gfCNCPoint2[15649] = {X 94.9398, Y 8.2871, Z -3.0000, A 0.000, B 0.000, C 0.000 }
gfCNCPoint2[15650] = {X 95.7852, Y 8.5829, Z -3.0000, A 0.000, B 0.000, C 0.000 }
gfCNCPoint2[15651] = {X 96.5436, Y 9.0595, Z -3.0000, A 0.000, B 0.000, C 0.000 }
gfCNCPoint2[15652] = {X 97.1770, Y 9.6929, Z -3.0000, A 0.000, B 0.000, C 0.000 }
gfCNCPoint2[15653] = {X 97.6535, Y 10.4513, Z -3.0000, A 0.000, B 0.000, C 0.000 }
gfCNCPoint2[15654] = {X 97.9494, Y 11.2967, Z -3.0000, A 0.000, B 0.000, C 0.000 }
gfCNCPoint2[15655] = {X 98.0497, Y 12.1868, Z -3.0000, A 0.000, B 0.000, C 0.000 }
gfCNCPoint2[15656] = {X 98.0495, Y 13.0192, Z -3.0000, A 0.000, B 0.000, C 0.000 }
gfCNCPoint2[15657] = {X 97.9794, Y 13.7247, Z -3.0000, A 0.000, B 0.000, C 0.000 }
gfCNCPoint2[15658] = {X 97.7858, Y 14.4068, Z -3.0000, A 0.000, B 0.000, C 0.000 }
gfCNCPoint2[15659] = {X 97.4749, Y 15.0440, Z -3.0000, A 0.000, B 0.000, C 0.000 }
gfCNCPoint2[15660] = {X 97.4127, Y 15.1437, Z -3.0000, A 0.000, B 0.000, C 0.000 }
gfCNCPoint2[15661] = {X 97.3476, Y 15.2415, Z -3.0000, A 0.000, B 0.000, C 0.000 }
gfCNCPoint2[15662] = {X 97.4105, Y 15.3108, Z -3.0000, A 0.000, B 0.000, C 0.000 }
gfCNCPoint2[15663] = {X 97.9961, Y 16.7687, Z -3.0000, A 0.000, B 0.000, C 0.000 }
gfCNCPoint2[15664] = {X 101.6269, Y 25.7689, Z -3.0000, A 0.000, B 0.000, C 0.000 }
gfCNCPoint2[15665] = {X 101.8768, Y 26.3801, Z -3.0000, A 0.000, B 0.000, C 0.000 }
gfCNCPoint2[15666] = {X 102.1268, Y 25.7689, Z -3.0000, A 0.000, B 0.000, C 0.000 }
gfCNCPoint2[15667] = {X 106.3426, Y 15.2553, Z -3.0000, A 0.000, B 0.000, C 0.000 }
gfCNCPoint2[15668] = {X 106.3813, Y 15.1986, Z -3.0000, A 0.000, B 0.000, C 0.000 }
gfCNCPoint2[15669] = {X 106.3236, Y 15.1097, Z -3.0000, A 0.000, B 0.000, C 0.000 }
gfCNCPoint2[15670] = {X 106.2684, Y 15.0194, Z -3.0000, A 0.000, B 0.000, C 0.000 }
gfCNCPoint2[15671] = {X 105.9605, Y 14.3760, Z -3.0000, A 0.000, B 0.000, C 0.000 }
gfCNCPoint2[15672] = {X 105.7718, Y 13.6883, Z -3.0000, A 0.000, B 0.000, C 0.000 }
gfCNCPoint2[15673] = {X 105.7083, Y 12.9779, Z -3.0000, A 0.000, B 0.000, C 0.000 }
gfCNCPoint2[15674] = {X 105.7083, Y 12.1868, Z -3.0000, A 0.000, B 0.000, C 0.000 }
gfCNCPoint2[15675] = {X 105.8086, Y 11.2967, Z -3.0000, A 0.000, B 0.000, C 0.000 }
gfCNCPoint2[15676] = {X 106.1044, Y 10.4513, Z -3.0000, A 0.000, B 0.000, C 0.000 }
gfCNCPoint2[15677] = {X 106.5810, Y 9.6929, Z -3.0000, A 0.000, B 0.000, C 0.000 }
gfCNCPoint2[15678] = {X 107.2143, Y 9.0595, Z -3.0000, A 0.000, B 0.000, C 0.000 }
gfCNCPoint2[15679] = {X 107.9727, Y 8.5829, Z -3.0000, A 0.000, B 0.000, C 0.000 }
gfCNCPoint2[15680] = {X 108.8182, Y 8.2871, Z -3.0000, A 0.000, B 0.000, C 0.000 }
gfCNCPoint2[15681] = {X 109.7083, Y 8.1868, Z -3.0000, A 0.000, B 0.000, C 0.000 }
gfCNCPoint2[15682] = {X 117.7916, Y 8.1868, Z -3.0000, A 0.000, B 0.000, C 0.000 }
gfCNCPoint2[15683] = {X 118.6817, Y 8.2871, Z -3.0000, A 0.000, B 0.000, C 0.000 }
gfCNCPoint2[15684] = {X 119.5271, Y 8.5829, Z -3.0000, A 0.000, B 0.000, C 0.000 }
gfCNCPoint2[15685] = {X 120.2855, Y 9.0595, Z -3.0000, A 0.000, B 0.000, C 0.000 }
gfCNCPoint2[15686] = {X 120.9189, Y 9.6929, Z -3.0000, A 0.000, B 0.000, C 0.000 }
gfCNCPoint2[15687] = {X 121.3955, Y 10.4513, Z -3.0000, A 0.000, B 0.000, C 0.000 }
gfCNCPoint2[15688] = {X 121.6913, Y 11.2967, Z -3.0000, A 0.000, B 0.000, C 0.000 }
gfCNCPoint2[15689] = {X 121.7916, Y 12.1868, Z -3.0000, A 0.000, B 0.000, C 0.000 }
gfCNCPoint2[15690] = {X 121.7914, Y 13.0192, Z -3.0000, A 0.000, B 0.000, C 0.000 }
gfCNCPoint2[15691] = {X 121.6828, Y 13.9047, Z -3.0000, A 0.000, B 0.000, C 0.000 }
gfCNCPoint2[15692] = {X 121.3806, Y 14.7440, Z -3.0000, A 0.000, B 0.000, C 0.000 }
gfCNCPoint2[15693] = {X 120.9000, Y 15.4955, Z -3.0000, A 0.000, B 0.000, C 0.000 }
gfCNCPoint2[15694] = {X 120.2647, Y 16.1219, Z -3.0000, A 0.000, B 0.000, C 0.000 }
gfCNCPoint2[15695] = {X 120.2634, Y 41.0662, Z -3.0000, A 0.000, B 0.000, C 0.000 }
gfCNCPoint2[15696] = {X 120.4160, Y 41.1901, Z -3.0000, A 0.000, B 0.000, C 0.000 }
gfCNCPoint2[15697] = {X 120.9967, Y 41.8157, Z -3.0000, A 0.000, B 0.000, C 0.000 }
gfCNCPoint2[15698] = {X 121.4315, Y 42.5502, Z -3.0000, A 0.000, B 0.000, C 0.000 }
gfCNCPoint2[15699] = {X 121.7005, Y 43.3602, Z -3.0000, A 0.000, B 0.000, C 0.000 }
gfCNCPoint2[15700] = {X 121.7916, Y 44.2089, Z -3.0000, A 0.000, B 0.000, C 0.000 }
gfCNCPoint2[15701] = {X 121.7916, Y 45.0000, Z -3.0000, A 0.000, B 0.000, C 0.000 }
gfCNCPoint2[15702] = {X 121.6913, Y 45.8901, Z -3.0000, A 0.000, B 0.000, C 0.000 }
gfCNCPoint2[15703] = {X 121.3955, Y 46.7355, Z -3.0000, A 0.000, B 0.000, C 0.000 }
gfCNCPoint2[15704] = {X 120.9189, Y 47.4940, Z -3.0000, A 0.000, B 0.000, C 0.000 }
gfCNCPoint2[15705] = {X 120.2855, Y 48.1273, Z -3.0000, A 0.000, B 0.000, C 0.000 }
gfCNCPoint2[15706] = {X 119.5271, Y 48.6039, Z -3.0000, A 0.000, B 0.000, C 0.000 }
gfCNCPoint2[15707] = {X 118.6817, Y 48.8997, Z -3.0000, A 0.000, B 0.000, C 0.000 }
gfCNCPoint2[15708] = {X 117.7916, Y 49.0000, Z -3.0000, A 0.000, B 0.000, C 0.000 }
gfCNCPoint2[15709] = {X 111.9185, Y 49.0000, Z -3.0000, A 0.000, B 0.000, C 0.000 }
gfCNCPoint2[15710] = {X 111.0284, Y 48.8997, Z -3.0000, A 0.000, B 0.000, C 0.000 }
gfCNCPoint2[15711] = {X 110.1829, Y 48.6039, Z -3.0000, A 0.000, B 0.000, C 0.000 }
gfCNCPoint2[15712] = {X 109.4245, Y 48.1273, Z -3.0000, A 0.000, B 0.000, C 0.000 }
gfCNCPoint2[15713] = {X 108.7911, Y 47.4939, Z -3.0000, A 0.000, B 0.000, C 0.000 }
gfCNCPoint2[15714] = {X 108.3146, Y 46.7355, Z -3.0000, A 0.000, B 0.000, C 0.000 }
gfCNCPoint2[15715] = {X 108.0188, Y 45.8900, Z -3.0000, A 0.000, B 0.000, C 0.000 }
gfCNCPoint2[15716] = {X 107.9185, Y 45.0000, Z -3.0000, A 0.000, B 0.000, C 0.000 }
gfCNCPoint2[15717] = {X 107.9185, Y 44.1811, Z -3.0000, A 0.000, B 0.000, C 0.000 }
gfCNCPoint2[15718] = {X 107.9517, Y 43.6776, Z -3.0000, A 0.000, B 0.000, C 0.000 }
gfCNCPoint2[15719] = {X 108.0507, Y 43.1827, Z -3.0000, A 0.000, B 0.000, C 0.000 }
gfCNCPoint2[15720] = {X 108.2043, Y 42.7280, Z -3.0000, A 0.000, B 0.000, C 0.000 }
gfCNCPoint2[15721] = {X 108.4135, Y 42.2960, Z -3.0000, A 0.000, B 0.000, C 0.000 }
gfCNCPoint2[15722] = {X 108.4390, Y 42.2514, Z -3.0000, A 0.000, B 0.000, C 0.000 }
gfCNCPoint2[15723] = {X 108.4651, Y 42.2073, Z -3.0000, A 0.000, B 0.000, C 0.000 }
gfCNCPoint2[15724] = {X 108.9129, Y 41.5686, Z -3.0000, A 0.000, B 0.000, C 0.000 }
gfCNCPoint2[15725] = {X 109.4466, Y 40.9999, Z -3.0000, A 0.000, B 0.000, C 0.000 }
gfCNCPoint2[15726] = {X 109.4465, Y 38.9229, Z -3.0000, A 0.000, B 0.000, C 0.000 }
gfCNCPoint2[15727] = {X 108.9328, Y 38.9229, Z -3.0000, A 0.000, B 0.000, C 0.000 }
gfCNCPoint2[15728] = {X 105.8164, Y 46.5384, Z -3.0000, A 0.000, B 0.000, C 0.000 }
gfCNCPoint2[15729] = {X 105.3339, Y 47.3869, Z -3.0000, A 0.000, B 0.000, C 0.000 }
gfCNCPoint2[15730] = {X 104.6602, Y 48.0932, Z -3.0000, A 0.000, B 0.000, C 0.000 }
gfCNCPoint2[15731] = {X 103.8355, Y 48.6154, Z -3.0000, A 0.000, B 0.000, C 0.000 }
gfCNCPoint2[15732] = {X 102.9580, Y 48.9121, Z -3.0000, A 0.000, B 0.000, C 0.000 }
gfCNCPoint2[15733] = {X 102.0357, Y 48.9990, Z -3.0000, A 0.000, B 0.000, C 0.000 }
gfCNCPoint2[15734] = {X 101.1182, Y 48.8715, Z -3.0000, A 0.000, B 0.000, C 0.000 }
gfCNCPoint2[15735] = {X 100.2546, Y 48.5362, Z -3.0000, A 0.000, B 0.000, C 0.000 }
gfCNCPoint2[15736] = {X 99.4912, Y 48.0114, Z -3.0000, A 0.000, B 0.000, C 0.000 }
gfCNCPoint2[15737] = {X 98.8691, Y 47.3250, Z -3.0000, A 0.000, B 0.000, C 0.000 }
gfCNCPoint2[15738] = {X 98.4216, Y 46.5139, Z -3.0000, A 0.000, B 0.000, C 0.000 }
gfCNCPoint2[15739] = {X 94.8150, Y 37.6933, Z -3.0000, A 0.000, B 0.000, C 0.000 }
gfCNCPoint2[15740] = {X 94.8103, Y 38.2306, Z -3.0000, A 0.000, B 0.000, C 0.000 }
gfCNCPoint2[15741] = {X 94.8105, Y 41.0553, Z -3.0000, A 0.000, B 0.000, C 0.000 }
gfCNCPoint2[15742] = {X 95.3658, Y 41.5952, Z -3.0000, A 0.000, B 0.000, C 0.000 }
gfCNCPoint2[15743] = {X 95.8092, Y 42.2301, Z -3.0000, A 0.000, B 0.000, C 0.000 }
gfCNCPoint2[15744] = {X 96.0347, Y 42.6952, Z -3.0000, A 0.000, B 0.000, C 0.000 }
gfCNCPoint2[15745] = {X 96.1997, Y 43.1852, Z -3.0000, A 0.000, B 0.000, C 0.000 }
gfCNCPoint2[15746] = {X 96.3016, Y 43.6926, Z -3.0000, A 0.000, B 0.000, C 0.000 }
gfCNCPoint2[15747] = {X 96.3385, Y 44.2089, Z -3.0000, A 0.000, B 0.000, C 0.000 }
gfCNCPoint2[15748] = {X 96.3384, Y 45.0384, Z -3.0000, A 0.000, B 0.000, C 0.000 }
gfCNCPoint2[15749] = {X 96.2308, Y 45.9222, Z -3.0000, A 0.000, B 0.000, C 0.000 }
gfCNCPoint2[15750] = {X 95.9304, Y 46.7602, Z -3.0000, A 0.000, B 0.000, C 0.000 }
gfCNCPoint2[15751] = {X 95.4521, Y 47.5111, Z -3.0000, A 0.000, B 0.000, C 0.000 }
gfCNCPoint2[15752] = {X 94.8196, Y 48.1376, Z -3.0000, A 0.000, B 0.000, C 0.000 }
gfCNCPoint2[15753] = {X 94.0642, Y 48.6086, Z -3.0000, A 0.000, B 0.000, C 0.000 }
gfCNCPoint2[15754] = {X 93.2233, Y 48.9009, Z -3.0000, A 0.000, B 0.000, C 0.000 }
gfCNCPoint2[15755] = {X 92.3385, Y 49.0000, Z -3.0000, A 0.000, B 0.000, C 0.000 }
gfCNCPoint2[15756] = {X 85.8951, Y 49.0000, Z -3.0000, A 0.000, B 0.000, C 0.000 }
gfCNCPoint2[15757] = {X 85.0050, Y 48.8997, Z -3.0000, A 0.000, B 0.000, C 0.000 }
gfCNCPoint2[15758] = {X 84.1595, Y 48.6039, Z -3.0000, A 0.000, B 0.000, C 0.000 }
gfCNCPoint2[15759] = {X 83.4011, Y 48.1273, Z -3.0000, A 0.000, B 0.000, C 0.000 }
gfCNCPoint2[15760] = {X 82.7677, Y 47.4939, Z -3.0000, A 0.000, B 0.000, C 0.000 }
gfCNCPoint2[15761] = {X 82.2912, Y 46.7355, Z -3.0000, A 0.000, B 0.000, C 0.000 }
gfCNCPoint2[15762] = {X 81.9954, Y 45.8900, Z -3.0000, A 0.000, B 0.000, C 0.000 }
gfCNCPoint2[15763] = {X 81.8951, Y 45.0000, Z -3.0000, A 0.000, B 0.000, C 0.000 }
gfCNCPoint2[15764] = {X 81.8951, Y 44.2089, Z -3.0000, A 0.000, B 0.000, C 0.000 }
gfCNCPoint2[15765] = {X 82.0011, Y 43.3123, Z -3.0000, A 0.000, B 0.000, C 0.000 }
gfCNCPoint2[15766] = {X 82.3025, Y 42.4613, Z -3.0000, A 0.000, B 0.000, C 0.000 }
gfCNCPoint2[15767] = {X 82.7846, Y 41.6979, Z -3.0000, A 0.000, B 0.000, C 0.000 }
gfCNCPoint2[15768] = {X 83.4234, Y 41.0598, Z -3.0000, A 0.000, B 0.000, C 0.000 }
gfCNCPoint2[15769] = {X 83.4233, Y 28.5920, Z -3.0000, A 0.000, B 0.000, C 0.000 }
gfCNCPoint2[15770] = {X 79.3433, Y 28.5920, Z -3.0000, A 0.000, B 0.000, C 0.000 }
gfCNCPoint2[15771] = {X 79.3433, Y 28.5920, Z 0.0000, A 0.000, B 0.000, C 0.000 }
gfCNCPoint2[15772] = {X 79.3433, Y 28.5920, Z 11.0000, A 0.000, B 0.000, C 0.000 }
gfCNCPoint2[15773] = {X 136.1636, Y 30.3963, Z 11.0000, A 0.000, B 0.000, C 0.000 }
gfCNCPoint2[15774] = {X 136.1636, Y 30.3963, Z 0.0000, A 0.000, B 0.000, C 0.000 }
gfCNCPoint2[15775] = {X 136.1636, Y 30.3963, Z -3.0000, A 0.000, B 0.000, C 0.000 }
gfCNCPoint2[15776] = {X 140.2436, Y 30.3963, Z -3.0000, A 0.000, B 0.000, C 0.000 }
gfCNCPoint2[15777] = {X 140.2436, Y 19.8770, Z -3.0000, A 0.000, B 0.000, C 0.000 }
gfCNCPoint2[15778] = {X 137.4242, Y 19.8766, Z -3.0000, A 0.000, B 0.000, C 0.000 }
gfCNCPoint2[15779] = {X 136.8918, Y 20.5215, Z -3.0000, A 0.000, B 0.000, C 0.000 }
gfCNCPoint2[15780] = {X 136.2452, Y 21.0516, Z -3.0000, A 0.000, B 0.000, C 0.000 }
gfCNCPoint2[15781] = {X 135.5085, Y 21.4473, Z -3.0000, A 0.000, B 0.000, C 0.000 }
gfCNCPoint2[15782] = {X 134.7094, Y 21.6936, Z -3.0000, A 0.000, B 0.000, C 0.000 }
gfCNCPoint2[15783] = {X 133.8778, Y 21.7814, Z -3.0000, A 0.000, B 0.000, C 0.000 }
gfCNCPoint2[15784] = {X 133.2006, Y 21.7815, Z -3.0000, A 0.000, B 0.000, C 0.000 }
gfCNCPoint2[15785] = {X 132.2394, Y 21.6732, Z -3.0000, A 0.000, B 0.000, C 0.000 }
gfCNCPoint2[15786] = {X 131.3263, Y 21.3537, Z -3.0000, A 0.000, B 0.000, C 0.000 }
gfCNCPoint2[15787] = {X 130.5072, Y 20.8390, Z -3.0000, A 0.000, B 0.000, C 0.000 }
gfCNCPoint2[15788] = {X 129.8231, Y 20.1550, Z -3.0000, A 0.000, B 0.000, C 0.000 }
gfCNCPoint2[15789] = {X 129.3085, Y 19.3359, Z -3.0000, A 0.000, B 0.000, C 0.000 }
gfCNCPoint2[15790] = {X 128.9890, Y 18.4228, Z -3.0000, A 0.000, B 0.000, C 0.000 }
gfCNCPoint2[15791] = {X 128.8806, Y 17.4615, Z -3.0000, A 0.000, B 0.000, C 0.000 }
gfCNCPoint2[15792] = {X 128.8806, Y 10.4835, Z -3.0000, A 0.000, B 0.000, C 0.000 }
gfCNCPoint2[15793] = {X 128.9874, Y 9.5289, Z -3.0000, A 0.000, B 0.000, C 0.000 }
gfCNCPoint2[15794] = {X 129.3026, Y 8.6214, Z -3.0000, A 0.000, B 0.000, C 0.000 }
gfCNCPoint2[15795] = {X 129.8104, Y 7.8061, Z -3.0000, A 0.000, B 0.000, C 0.000 }
gfCNCPoint2[15796] = {X 130.4859, Y 7.1231, Z -3.0000, A 0.000, B 0.000, C 0.000 }
gfCNCPoint2[15797] = {X 131.2956, Y 6.6063, Z -3.0000, A 0.000, B 0.000, C 0.000 }
gfCNCPoint2[15798] = {X 132.1995, Y 6.2811, Z -3.0000, A 0.000, B 0.000, C 0.000 }
gfCNCPoint2[15799] = {X 133.1529, Y 6.1638, Z -3.0000, A 0.000, B 0.000, C 0.000 }
gfCNCPoint2[15800] = {X 133.8866, Y 6.1637, Z -3.0000, A 0.000, B 0.000, C 0.000 }
gfCNCPoint2[15801] = {X 134.7112, Y 6.2518, Z -3.0000, A 0.000, B 0.000, C 0.000 }
gfCNCPoint2[15802] = {X 135.5038, Y 6.4958, Z -3.0000, A 0.000, B 0.000, C 0.000 }
gfCNCPoint2[15803] = {X 136.2352, Y 6.8868, Z -3.0000, A 0.000, B 0.000, C 0.000 }
gfCNCPoint2[15804] = {X 136.8784, Y 7.4103, Z -3.0000, A 0.000, B 0.000, C 0.000 }
gfCNCPoint2[15805] = {X 137.4097, Y 8.0470, Z -3.0000, A 0.000, B 0.000, C 0.000 }
gfCNCPoint2[15806] = {X 155.1123, Y 8.0482, Z -3.0000, A 0.000, B 0.000, C 0.000 }
gfCNCPoint2[15807] = {X 155.6443, Y 7.4103, Z -3.0000, A 0.000, B 0.000, C 0.000 }
gfCNCPoint2[15808] = {X 156.2886, Y 6.8861, Z -3.0000, A 0.000, B 0.000, C 0.000 }
gfCNCPoint2[15809] = {X 157.0212, Y 6.4948, Z -3.0000, A 0.000, B 0.000, C 0.000 }
gfCNCPoint2[15810] = {X 157.8152, Y 6.2510, Z -3.0000, A 0.000, B 0.000, C 0.000 }
gfCNCPoint2[15811] = {X 158.6412, Y 6.1637, Z -3.0000, A 0.000, B 0.000, C 0.000 }
gfCNCPoint2[15812] = {X 159.3781, Y 6.1639, Z -3.0000, A 0.000, B 0.000, C 0.000 }
gfCNCPoint2[15813] = {X 160.3301, Y 6.2828, Z -3.0000, A 0.000, B 0.000, C 0.000 }
gfCNCPoint2[15814] = {X 161.2324, Y 6.6088, Z -3.0000, A 0.000, B 0.000, C 0.000 }
gfCNCPoint2[15815] = {X 162.0405, Y 7.1260, Z -3.0000, A 0.000, B 0.000, C 0.000 }
gfCNCPoint2[15816] = {X 162.7145, Y 7.8088, Z -3.0000, A 0.000, B 0.000, C 0.000 }
gfCNCPoint2[15817] = {X 163.2212, Y 8.6236, Z -3.0000, A 0.000, B 0.000, C 0.000 }
gfCNCPoint2[15818] = {X 163.5355, Y 9.5300, Z -3.0000, A 0.000, B 0.000, C 0.000 }
gfCNCPoint2[15819] = {X 163.6421, Y 10.4835, Z -3.0000, A 0.000, B 0.000, C 0.000 }
gfCNCPoint2[15820] = {X 163.6421, Y 17.4615, Z -3.0000, A 0.000, B 0.000, C 0.000 }
gfCNCPoint2[15821] = {X 163.5355, Y 18.4152, Z -3.0000, A 0.000, B 0.000, C 0.000 }
gfCNCPoint2[15822] = {X 163.2211, Y 19.3218, Z -3.0000, A 0.000, B 0.000, C 0.000 }
gfCNCPoint2[15823] = {X 162.7142, Y 20.1366, Z -3.0000, A 0.000, B 0.000, C 0.000 }
gfCNCPoint2[15824] = {X 162.0400, Y 20.8194, Z -3.0000, A 0.000, B 0.000, C 0.000 }
gfCNCPoint2[15825] = {X 161.2318, Y 21.3365, Z -3.0000, A 0.000, B 0.000, C 0.000 }
gfCNCPoint2[15826] = {X 160.3292, Y 21.6625, Z -3.0000, A 0.000, B 0.000, C 0.000 }
gfCNCPoint2[15827] = {X 159.3770, Y 21.7812, Z -3.0000, A 0.000, B 0.000, C 0.000 }
gfCNCPoint2[15828] = {X 158.6791, Y 21.7815, Z -3.0000, A 0.000, B 0.000, C 0.000 }
gfCNCPoint2[15829] = {X 157.8408, Y 21.6961, Z -3.0000, A 0.000, B 0.000, C 0.000 }
gfCNCPoint2[15830] = {X 157.0346, Y 21.4510, Z -3.0000, A 0.000, B 0.000, C 0.000 }
gfCNCPoint2[15831] = {X 156.2906, Y 21.0553, Z -3.0000, A 0.000, B 0.000, C 0.000 }
gfCNCPoint2[15832] = {X 155.6368, Y 20.5237, Z -3.0000, A 0.000, B 0.000, C 0.000 }
gfCNCPoint2[15833] = {X 155.0975, Y 19.8763, Z -3.0000, A 0.000, B 0.000, C 0.000 }
gfCNCPoint2[15834] = {X 152.2760, Y 19.8776, Z -3.0000, A 0.000, B 0.000, C 0.000 }
gfCNCPoint2[15835] = {X 152.2744, Y 40.8742, Z -3.0000, A 0.000, B 0.000, C 0.000 }
gfCNCPoint2[15836] = {X 152.7409, Y 41.3763, Z -3.0000, A 0.000, B 0.000, C 0.000 }
gfCNCPoint2[15837] = {X 152.8353, Y 41.4889, Z -3.0000, A 0.000, B 0.000, C 0.000 }
gfCNCPoint2[15838] = {X 153.3607, Y 42.3142, Z -3.0000, A 0.000, B 0.000, C 0.000 }
gfCNCPoint2[15839] = {X 153.6888, Y 43.2358, Z -3.0000, A 0.000, B 0.000, C 0.000 }
gfCNCPoint2[15840] = {X 153.8031, Y 44.2074, Z -3.0000, A 0.000, B 0.000, C 0.000 }
gfCNCPoint2[15841] = {X 153.8029, Y 45.0415, Z -3.0000, A 0.000, B 0.000, C 0.000 }
gfCNCPoint2[15842] = {X 153.6867, Y 45.9960, Z -3.0000, A 0.000, B 0.000, C 0.000 }
gfCNCPoint2[15843] = {X 153.3623, Y 46.9011, Z -3.0000, A 0.000, B 0.000, C 0.000 }
gfCNCPoint2[15844] = {X 152.8458, Y 47.7120, Z -3.0000, A 0.000, B 0.000, C 0.000 }
gfCNCPoint2[15845] = {X 152.1626, Y 48.3886, Z -3.0000, A 0.000, B 0.000, C 0.000 }
gfCNCPoint2[15846] = {X 151.3468, Y 48.8973, Z -3.0000, A 0.000, B 0.000, C 0.000 }
gfCNCPoint2[15847] = {X 150.4386, Y 49.2130, Z -3.0000, A 0.000, B 0.000, C 0.000 }
gfCNCPoint2[15848] = {X 149.4831, Y 49.3200, Z -3.0000, A 0.000, B 0.000, C 0.000 }
gfCNCPoint2[15849] = {X 143.0396, Y 49.3200, Z -3.0000, A 0.000, B 0.000, C 0.000 }
gfCNCPoint2[15850] = {X 142.0831, Y 49.2128, Z -3.0000, A 0.000, B 0.000, C 0.000 }
gfCNCPoint2[15851] = {X 141.1741, Y 48.8964, Z -3.0000, A 0.000, B 0.000, C 0.000 }
gfCNCPoint2[15852] = {X 140.3576, Y 48.3866, Z -3.0000, A 0.000, B 0.000, C 0.000 }
gfCNCPoint2[15853] = {X 139.6743, Y 47.7087, Z -3.0000, A 0.000, B 0.000, C 0.000 }
gfCNCPoint2[15854] = {X 139.1581, Y 46.8964, Z -3.0000, A 0.000, B 0.000, C 0.000 }
gfCNCPoint2[15855] = {X 138.8346, Y 45.9899, Z -3.0000, A 0.000, B 0.000, C 0.000 }
gfCNCPoint2[15856] = {X 138.7198, Y 45.0342, Z -3.0000, A 0.000, B 0.000, C 0.000 }
gfCNCPoint2[15857] = {X 138.7200, Y 44.1494, Z -3.0000, A 0.000, B 0.000, C 0.000 }
gfCNCPoint2[15858] = {X 138.8305, Y 43.2364, Z -3.0000, A 0.000, B 0.000, C 0.000 }
gfCNCPoint2[15859] = {X 139.1317, Y 42.3675, Z -3.0000, A 0.000, B 0.000, C 0.000 }
gfCNCPoint2[15860] = {X 139.6099, Y 41.5821, Z -3.0000, A 0.000, B 0.000, C 0.000 }
gfCNCPoint2[15861] = {X 140.2436, Y 40.9157, Z -3.0000, A 0.000, B 0.000, C 0.000 }
gfCNCPoint2[15862] = {X 140.2436, Y 30.3963, Z -3.0000, A 0.000, B 0.000, C 0.000 }
gfCNCPoint2[15863] = {X 136.2436, Y 30.3963, Z -3.0000, A 0.000, B 0.000, C 0.000 }
gfCNCPoint2[15864] = {X 140.3236, Y 30.3963, Z -3.0000, A 0.000, B 0.000, C 0.000 }
gfCNCPoint2[15865] = {X 140.3236, Y 19.7970, Z -3.0000, A 0.000, B 0.000, C 0.000 }
gfCNCPoint2[15866] = {X 137.3799, Y 19.7962, Z -3.0000, A 0.000, B 0.000, C 0.000 }
gfCNCPoint2[15867] = {X 137.3570, Y 19.8332, Z -3.0000, A 0.000, B 0.000, C 0.000 }
gfCNCPoint2[15868] = {X 136.8345, Y 20.4656, Z -3.0000, A 0.000, B 0.000, C 0.000 }
gfCNCPoint2[15869] = {X 136.1999, Y 20.9857, Z -3.0000, A 0.000, B 0.000, C 0.000 }
gfCNCPoint2[15870] = {X 135.4771, Y 21.3737, Z -3.0000, A 0.000, B 0.000, C 0.000 }
gfCNCPoint2[15871] = {X 134.6930, Y 21.6153, Z -3.0000, A 0.000, B 0.000, C 0.000 }
gfCNCPoint2[15872] = {X 133.8772, Y 21.7014, Z -3.0000, A 0.000, B 0.000, C 0.000 }
gfCNCPoint2[15873] = {X 133.2006, Y 21.7015, Z -3.0000, A 0.000, B 0.000, C 0.000 }
gfCNCPoint2[15874] = {X 132.2572, Y 21.5952, Z -3.0000, A 0.000, B 0.000, C 0.000 }
gfCNCPoint2[15875] = {X 131.3610, Y 21.2816, Z -3.0000, A 0.000, B 0.000, C 0.000 }
gfCNCPoint2[15876] = {X 130.5570, Y 20.7765, Z -3.0000, A 0.000, B 0.000, C 0.000 }
gfCNCPoint2[15877] = {X 129.8857, Y 20.1051, Z -3.0000, A 0.000, B 0.000, C 0.000 }
gfCNCPoint2[15878] = {X 129.3805, Y 19.3012, Z -3.0000, A 0.000, B 0.000, C 0.000 }
gfCNCPoint2[15879] = {X 129.0669, Y 18.4050, Z -3.0000, A 0.000, B 0.000, C 0.000 }
gfCNCPoint2[15880] = {X 128.9606, Y 17.4615, Z -3.0000, A 0.000, B 0.000, C 0.000 }
gfCNCPoint2[15881] = {X 128.9606, Y 10.4835, Z -3.0000, A 0.000, B 0.000, C 0.000 }
gfCNCPoint2[15882] = {X 129.0655, Y 9.5466, Z -3.0000, A 0.000, B 0.000, C 0.000 }
gfCNCPoint2[15883] = {X 129.3747, Y 8.6559, Z -3.0000, A 0.000, B 0.000, C 0.000 }
gfCNCPoint2[15884] = {X 129.8732, Y 7.8557, Z -3.0000, A 0.000, B 0.000, C 0.000 }
gfCNCPoint2[15885] = {X 130.5362, Y 7.1853, Z -3.0000, A 0.000, B 0.000, C 0.000 }
gfCNCPoint2[15886] = {X 131.3309, Y 6.6781, Z -3.0000, A 0.000, B 0.000, C 0.000 }
gfCNCPoint2[15887] = {X 132.2180, Y 6.3589, Z -3.0000, A 0.000, B 0.000, C 0.000 }
gfCNCPoint2[15888] = {X 133.1538, Y 6.2438, Z -3.0000, A 0.000, B 0.000, C 0.000 }
gfCNCPoint2[15889] = {X 133.8858, Y 6.2437, Z -3.0000, A 0.000, B 0.000, C 0.000 }
gfCNCPoint2[15890] = {X 134.7034, Y 6.3319, Z -3.0000, A 0.000, B 0.000, C 0.000 }
gfCNCPoint2[15891] = {X 135.4886, Y 6.5762, Z -3.0000, A 0.000, B 0.000, C 0.000 }
gfCNCPoint2[15892] = {X 136.2118, Y 6.9674, Z -3.0000, A 0.000, B 0.000, C 0.000 }
gfCNCPoint2[15893] = {X 136.8460, Y 7.4909, Z -3.0000, A 0.000, B 0.000, C 0.000 }
gfCNCPoint2[15894] = {X 137.3672, Y 8.1270, Z -3.0000, A 0.000, B 0.000, C 0.000 }
gfCNCPoint2[15895] = {X 155.1548, Y 8.1282, Z -3.0000, A 0.000, B 0.000, C 0.000 }
gfCNCPoint2[15896] = {X 155.6767, Y 7.4910, Z -3.0000, A 0.000, B 0.000, C 0.000 }
gfCNCPoint2[15897] = {X 156.3119, Y 6.9668, Z -3.0000, A 0.000, B 0.000, C 0.000 }
gfCNCPoint2[15898] = {X 157.0364, Y 6.5752, Z -3.0000, A 0.000, B 0.000, C 0.000 }
gfCNCPoint2[15899] = {X 157.8230, Y 6.3311, Z -3.0000, A 0.000, B 0.000, C 0.000 }
gfCNCPoint2[15900] = {X 158.6420, Y 6.2437, Z -3.0000, A 0.000, B 0.000, C 0.000 }
gfCNCPoint2[15901] = {X 159.3770, Y 6.2439, Z -3.0000, A 0.000, B 0.000, C 0.000 }
gfCNCPoint2[15902] = {X 160.3114, Y 6.3606, Z -3.0000, A 0.000, B 0.000, C 0.000 }
gfCNCPoint2[15903] = {X 161.1970, Y 6.6806, Z -3.0000, A 0.000, B 0.000, C 0.000 }
gfCNCPoint2[15904] = {X 161.9902, Y 7.1882, Z -3.0000, A 0.000, B 0.000, C 0.000 }
gfCNCPoint2[15905] = {X 162.6517, Y 7.8584, Z -3.0000, A 0.000, B 0.000, C 0.000 }
gfCNCPoint2[15906] = {X 163.1490, Y 8.6580, Z -3.0000, A 0.000, B 0.000, C 0.000 }
gfCNCPoint2[15907] = {X 163.4575, Y 9.5477, Z -3.0000, A 0.000, B 0.000, C 0.000 }
gfCNCPoint2[15908] = {X 163.5621, Y 10.4835, Z -3.0000, A 0.000, B 0.000, C 0.000 }
gfCNCPoint2[15909] = {X 163.5621, Y 17.4615, Z -3.0000, A 0.000, B 0.000, C 0.000 }
gfCNCPoint2[15910] = {X 163.4575, Y 18.3975, Z -3.0000, A 0.000, B 0.000, C 0.000 }
gfCNCPoint2[15911] = {X 163.1489, Y 19.2873, Z -3.0000, A 0.000, B 0.000, C 0.000 }
gfCNCPoint2[15912] = {X 162.6514, Y 20.0870, Z -3.0000, A 0.000, B 0.000, C 0.000 }
gfCNCPoint2[15913] = {X 161.9897, Y 20.7572, Z -3.0000, A 0.000, B 0.000, C 0.000 }
gfCNCPoint2[15914] = {X 161.1964, Y 21.2648, Z -3.0000, A 0.000, B 0.000, C 0.000 }
gfCNCPoint2[15915] = {X 160.3106, Y 21.5847, Z -3.0000, A 0.000, B 0.000, C 0.000 }
gfCNCPoint2[15916] = {X 159.3760, Y 21.7012, Z -3.0000, A 0.000, B 0.000, C 0.000 }
gfCNCPoint2[15917] = {X 158.6794, Y 21.7015, Z -3.0000, A 0.000, B 0.000, C 0.000 }
gfCNCPoint2[15918] = {X 157.8482, Y 21.6160, Z -3.0000, A 0.000, B 0.000, C 0.000 }
gfCNCPoint2[15919] = {X 157.0495, Y 21.3706, Z -3.0000, A 0.000, B 0.000, C 0.000 }
gfCNCPoint2[15920] = {X 156.3138, Y 20.9745, Z -3.0000, A 0.000, B 0.000, C 0.000 }
gfCNCPoint2[15921] = {X 155.6691, Y 20.4430, Z -3.0000, A 0.000, B 0.000, C 0.000 }
gfCNCPoint2[15922] = {X 155.1400, Y 19.7963, Z -3.0000, A 0.000, B 0.000, C 0.000 }
gfCNCPoint2[15923] = {X 152.1960, Y 19.7977, Z -3.0000, A 0.000, B 0.000, C 0.000 }
gfCNCPoint2[15924] = {X 152.1944, Y 40.9056, Z -3.0000, A 0.000, B 0.000, C 0.000 }
gfCNCPoint2[15925] = {X 152.6809, Y 41.4293, Z -3.0000, A 0.000, B 0.000, C 0.000 }
gfCNCPoint2[15926] = {X 152.7735, Y 41.5398, Z -3.0000, A 0.000, B 0.000, C 0.000 }
gfCNCPoint2[15927] = {X 153.2890, Y 42.3497, Z -3.0000, A 0.000, B 0.000, C 0.000 }
gfCNCPoint2[15928] = {X 153.6109, Y 43.2542, Z -3.0000, A 0.000, B 0.000, C 0.000 }
gfCNCPoint2[15929] = {X 153.7231, Y 44.2078, Z -3.0000, A 0.000, B 0.000, C 0.000 }
gfCNCPoint2[15930] = {X 153.7229, Y 45.0408, Z -3.0000, A 0.000, B 0.000, C 0.000 }
gfCNCPoint2[15931] = {X 153.6089, Y 45.9775, Z -3.0000, A 0.000, B 0.000, C 0.000 }
gfCNCPoint2[15932] = {X 153.2905, Y 46.8659, Z -3.0000, A 0.000, B 0.000, C 0.000 }
gfCNCPoint2[15933] = {X 152.7835, Y 47.6618, Z -3.0000, A 0.000, B 0.000, C 0.000 }
gfCNCPoint2[15934] = {X 152.1130, Y 48.3258, Z -3.0000, A 0.000, B 0.000, C 0.000 }
gfCNCPoint2[15935] = {X 151.3123, Y 48.8251, Z -3.0000, A 0.000, B 0.000, C 0.000 }
gfCNCPoint2[15936] = {X 150.4209, Y 49.1350, Z -3.0000, A 0.000, B 0.000, C 0.000 }
gfCNCPoint2[15937] = {X 149.4831, Y 49.2400, Z -3.0000, A 0.000, B 0.000, C 0.000 }
gfCNCPoint2[15938] = {X 143.0396, Y 49.2400, Z -3.0000, A 0.000, B 0.000, C 0.000 }
gfCNCPoint2[15939] = {X 142.1008, Y 49.1348, Z -3.0000, A 0.000, B 0.000, C 0.000 }
gfCNCPoint2[15940] = {X 141.2086, Y 48.8243, Z -3.0000, A 0.000, B 0.000, C 0.000 }
gfCNCPoint2[15941] = {X 140.4073, Y 48.3239, Z -3.0000, A 0.000, B 0.000, C 0.000 }
gfCNCPoint2[15942] = {X 139.7367, Y 47.6586, Z -3.0000, A 0.000, B 0.000, C 0.000 }
gfCNCPoint2[15943] = {X 139.2300, Y 46.8612, Z -3.0000, A 0.000, B 0.000, C 0.000 }
gfCNCPoint2[15944] = {X 138.9124, Y 45.9715, Z -3.0000, A 0.000, B 0.000, C 0.000 }
gfCNCPoint2[15945] = {X 138.7998, Y 45.0336, Z -3.0000, A 0.000, B 0.000, C 0.000 }
gfCNCPoint2[15946] = {X 138.8000, Y 44.1505, Z -3.0000, A 0.000, B 0.000, C 0.000 }
gfCNCPoint2[15947] = {X 138.9105, Y 43.2454, Z -3.0000, A 0.000, B 0.000, C 0.000 }
gfCNCPoint2[15948] = {X 139.2119, Y 42.3850, Z -3.0000, A 0.000, B 0.000, C 0.000 }
gfCNCPoint2[15949] = {X 139.6903, Y 41.6088, Z -3.0000, A 0.000, B 0.000, C 0.000 }
gfCNCPoint2[15950] = {X 140.3236, Y 40.9529, Z -3.0000, A 0.000, B 0.000, C 0.000 }
gfCNCPoint2[15951] = {X 140.3236, Y 30.3963, Z -3.0000, A 0.000, B 0.000, C 0.000 }
gfCNCPoint2[15952] = {X 136.3236, Y 30.3963, Z -3.0000, A 0.000, B 0.000, C 0.000 }
gfCNCPoint2[15953] = {X 140.4036, Y 30.3963, Z -3.0000, A 0.000, B 0.000, C 0.000 }
gfCNCPoint2[15954] = {X 140.4036, Y 19.7170, Z -3.0000, A 0.000, B 0.000, C 0.000 }
gfCNCPoint2[15955] = {X 137.3354, Y 19.7162, Z -3.0000, A 0.000, B 0.000, C 0.000 }
gfCNCPoint2[15956] = {X 137.2898, Y 19.7897, Z -3.0000, A 0.000, B 0.000, C 0.000 }
gfCNCPoint2[15957] = {X 136.7771, Y 20.4098, Z -3.0000, A 0.000, B 0.000, C 0.000 }
gfCNCPoint2[15958] = {X 136.1547, Y 20.9197, Z -3.0000, A 0.000, B 0.000, C 0.000 }
gfCNCPoint2[15959] = {X 135.4457, Y 21.3001, Z -3.0000, A 0.000, B 0.000, C 0.000 }
gfCNCPoint2[15960] = {X 134.6767, Y 21.5370, Z -3.0000, A 0.000, B 0.000, C 0.000 }
gfCNCPoint2[15961] = {X 133.8765, Y 21.6214, Z -3.0000, A 0.000, B 0.000, C 0.000 }
gfCNCPoint2[15962] = {X 133.2006, Y 21.6215, Z -3.0000, A 0.000, B 0.000, C 0.000 }
gfCNCPoint2[15963] = {X 132.2750, Y 21.5172, Z -3.0000, A 0.000, B 0.000, C 0.000 }
gfCNCPoint2[15964] = {X 131.3957, Y 21.2096, Z -3.0000, A 0.000, B 0.000, C 0.000 }
gfCNCPoint2[15965] = {X 130.6069, Y 20.7140, Z -3.0000, A 0.000, B 0.000, C 0.000 }
gfCNCPoint2[15966] = {X 129.9482, Y 20.0553, Z -3.0000, A 0.000, B 0.000, C 0.000 }
gfCNCPoint2[15967] = {X 129.4526, Y 19.2665, Z -3.0000, A 0.000, B 0.000, C 0.000 }
gfCNCPoint2[15968] = {X 129.1449, Y 18.3872, Z -3.0000, A 0.000, B 0.000, C 0.000 }
gfCNCPoint2[15969] = {X 129.0406, Y 17.4615, Z -3.0000, A 0.000, B 0.000, C 0.000 }
gfCNCPoint2[15970] = {X 129.0406, Y 10.4835, Z -3.0000, A 0.000, B 0.000, C 0.000 }
gfCNCPoint2[15971] = {X 129.1435, Y 9.5642, Z -3.0000, A 0.000, B 0.000, C 0.000 }
gfCNCPoint2[15972] = {X 129.4469, Y 8.6904, Z -3.0000, A 0.000, B 0.000, C 0.000 }
gfCNCPoint2[15973] = {X 129.9360, Y 7.9052, Z -3.0000, A 0.000, B 0.000, C 0.000 }
gfCNCPoint2[15974] = {X 130.5864, Y 7.2475, Z -3.0000, A 0.000, B 0.000, C 0.000 }
gfCNCPoint2[15975] = {X 131.3661, Y 6.7499, Z -3.0000, A 0.000, B 0.000, C 0.000 }
gfCNCPoint2[15976] = {X 132.2366, Y 6.4368, Z -3.0000, A 0.000, B 0.000, C 0.000 }
gfCNCPoint2[15977] = {X 133.1547, Y 6.3238, Z -3.0000, A 0.000, B 0.000, C 0.000 }
gfCNCPoint2[15978] = {X 133.8850, Y 6.3237, Z -3.0000, A 0.000, B 0.000, C 0.000 }
gfCNCPoint2[15979] = {X 134.6955, Y 6.4119, Z -3.0000, A 0.000, B 0.000, C 0.000 }
gfCNCPoint2[15980] = {X 135.4732, Y 6.6565, Z -3.0000, A 0.000, B 0.000, C 0.000 }
gfCNCPoint2[15981] = {X 136.1883, Y 7.0481, Z -3.0000, A 0.000, B 0.000, C 0.000 }
gfCNCPoint2[15982] = {X 136.8133, Y 7.5716, Z -3.0000, A 0.000, B 0.000, C 0.000 }
gfCNCPoint2[15983] = {X 137.3241, Y 8.2070, Z -3.0000, A 0.000, B 0.000, C 0.000 }
gfCNCPoint2[15984] = {X 155.1978, Y 8.2082, Z -3.0000, A 0.000, B 0.000, C 0.000 }
gfCNCPoint2[15985] = {X 155.7094, Y 7.5717, Z -3.0000, A 0.000, B 0.000, C 0.000 }
gfCNCPoint2[15986] = {X 156.3354, Y 7.0475, Z -3.0000, A 0.000, B 0.000, C 0.000 }
gfCNCPoint2[15987] = {X 157.0517, Y 6.6556, Z -3.0000, A 0.000, B 0.000, C 0.000 }
gfCNCPoint2[15988] = {X 157.8308, Y 6.4112, Z -3.0000, A 0.000, B 0.000, C 0.000 }
gfCNCPoint2[15989] = {X 158.6427, Y 6.3237, Z -3.0000, A 0.000, B 0.000, C 0.000 }
gfCNCPoint2[15990] = {X 159.3760, Y 6.3239, Z -3.0000, A 0.000, B 0.000, C 0.000 }
gfCNCPoint2[15991] = {X 160.2928, Y 6.4383, Z -3.0000, A 0.000, B 0.000, C 0.000 }
gfCNCPoint2[15992] = {X 161.1617, Y 6.7524, Z -3.0000, A 0.000, B 0.000, C 0.000 }
gfCNCPoint2[15993] = {X 161.9398, Y 7.2504, Z -3.0000, A 0.000, B 0.000, C 0.000 }
gfCNCPoint2[15994] = {X 162.5889, Y 7.9079, Z -3.0000, A 0.000, B 0.000, C 0.000 }
gfCNCPoint2[15995] = {X 163.0768, Y 8.6925, Z -3.0000, A 0.000, B 0.000, C 0.000 }
gfCNCPoint2[15996] = {X 163.3795, Y 9.5653, Z -3.0000, A 0.000, B 0.000, C 0.000 }
gfCNCPoint2[15997] = {X 163.4821, Y 10.4835, Z -3.0000, A 0.000, B 0.000, C 0.000 }
gfCNCPoint2[15998] = {X 163.4821, Y 17.4615, Z -3.0000, A 0.000, B 0.000, C 0.000 }
gfCNCPoint2[15999] = {X 163.3795, Y 18.3798, Z -3.0000, A 0.000, B 0.000, C 0.000 }
gfCNCPoint2[16000] = {X 163.0767, Y 19.2527, Z -3.0000, A 0.000, B 0.000, C 0.000 }
gfCNCPoint2[16001] = {X 162.5887, Y 20.0373, Z -3.0000, A 0.000, B 0.000, C 0.000 }
gfCNCPoint2[16002] = {X 161.9396, Y 20.6948, Z -3.0000, A 0.000, B 0.000, C 0.000 }
gfCNCPoint2[16003] = {X 161.1613, Y 21.1929, Z -3.0000, A 0.000, B 0.000, C 0.000 }
gfCNCPoint2[16004] = {X 160.2923, Y 21.5068, Z -3.0000, A 0.000, B 0.000, C 0.000 }
gfCNCPoint2[16005] = {X 159.3755, Y 21.6212, Z -3.0000, A 0.000, B 0.000, C 0.000 }
gfCNCPoint2[16006] = {X 158.6798, Y 21.6215, Z -3.0000, A 0.000, B 0.000, C 0.000 }
gfCNCPoint2[16007] = {X 157.8558, Y 21.5359, Z -3.0000, A 0.000, B 0.000, C 0.000 }
gfCNCPoint2[16008] = {X 157.0647, Y 21.2902, Z -3.0000, A 0.000, B 0.000, C 0.000 }
gfCNCPoint2[16009] = {X 156.3372, Y 20.8938, Z -3.0000, A 0.000, B 0.000, C 0.000 }
gfCNCPoint2[16010] = {X 155.7017, Y 20.3622, Z -3.0000, A 0.000, B 0.000, C 0.000 }
gfCNCPoint2[16011] = {X 155.1831, Y 19.7162, Z -3.0000, A 0.000, B 0.000, C 0.000 }
gfCNCPoint2[16012] = {X 152.1160, Y 19.7177, Z -3.0000, A 0.000, B 0.000, C 0.000 }
gfCNCPoint2[16013] = {X 152.1144, Y 40.9370, Z -3.0000, A 0.000, B 0.000, C 0.000 }
gfCNCPoint2[16014] = {X 152.6209, Y 41.4822, Z -3.0000, A 0.000, B 0.000, C 0.000 }
gfCNCPoint2[16015] = {X 152.7117, Y 41.5906, Z -3.0000, A 0.000, B 0.000, C 0.000 }
gfCNCPoint2[16016] = {X 153.2173, Y 42.3853, Z -3.0000, A 0.000, B 0.000, C 0.000 }
gfCNCPoint2[16017] = {X 153.5331, Y 43.2727, Z -3.0000, A 0.000, B 0.000, C 0.000 }
gfCNCPoint2[16018] = {X 153.6431, Y 44.2082, Z -3.0000, A 0.000, B 0.000, C 0.000 }
gfCNCPoint2[16019] = {X 153.6429, Y 45.0400, Z -3.0000, A 0.000, B 0.000, C 0.000 }
gfCNCPoint2[16020] = {X 153.5310, Y 45.9591, Z -3.0000, A 0.000, B 0.000, C 0.000 }
gfCNCPoint2[16021] = {X 153.2186, Y 46.8306, Z -3.0000, A 0.000, B 0.000, C 0.000 }
gfCNCPoint2[16022] = {X 152.7212, Y 47.6115, Z -3.0000, A 0.000, B 0.000, C 0.000 }
gfCNCPoint2[16023] = {X 152.0634, Y 48.2631, Z -3.0000, A 0.000, B 0.000, C 0.000 }
gfCNCPoint2[16024] = {X 151.2778, Y 48.7530, Z -3.0000, A 0.000, B 0.000, C 0.000 }
gfCNCPoint2[16025] = {X 150.4032, Y 49.0570, Z -3.0000, A 0.000, B 0.000, C 0.000 }
gfCNCPoint2[16026] = {X 149.4831, Y 49.1600, Z -3.0000, A 0.000, B 0.000, C 0.000 }
gfCNCPoint2[16027] = {X 143.0396, Y 49.1600, Z -3.0000, A 0.000, B 0.000, C 0.000 }
gfCNCPoint2[16028] = {X 142.1185, Y 49.0567, Z -3.0000, A 0.000, B 0.000, C 0.000 }
gfCNCPoint2[16029] = {X 141.2432, Y 48.7521, Z -3.0000, A 0.000, B 0.000, C 0.000 }
gfCNCPoint2[16030] = {X 140.4570, Y 48.2612, Z -3.0000, A 0.000, B 0.000, C 0.000 }
gfCNCPoint2[16031] = {X 139.7990, Y 47.6084, Z -3.0000, A 0.000, B 0.000, C 0.000 }
gfCNCPoint2[16032] = {X 139.3019, Y 46.8261, Z -3.0000, A 0.000, B 0.000, C 0.000 }
gfCNCPoint2[16033] = {X 138.9903, Y 45.9532, Z -3.0000, A 0.000, B 0.000, C 0.000 }
gfCNCPoint2[16034] = {X 138.8798, Y 45.0329, Z -3.0000, A 0.000, B 0.000, C 0.000 }
gfCNCPoint2[16035] = {X 138.8800, Y 44.1516, Z -3.0000, A 0.000, B 0.000, C 0.000 }
gfCNCPoint2[16036] = {X 138.9906, Y 43.2545, Z -3.0000, A 0.000, B 0.000, C 0.000 }
gfCNCPoint2[16037] = {X 139.2922, Y 42.4026, Z -3.0000, A 0.000, B 0.000, C 0.000 }
gfCNCPoint2[16038] = {X 139.7708, Y 41.6358, Z -3.0000, A 0.000, B 0.000, C 0.000 }
gfCNCPoint2[16039] = {X 140.4036, Y 40.9906, Z -3.0000, A 0.000, B 0.000, C 0.000 }
gfCNCPoint2[16040] = {X 140.4036, Y 30.3963, Z -3.0000, A 0.000, B 0.000, C 0.000 }
gfCNCPoint2[16041] = {X 136.4036, Y 30.3963, Z -3.0000, A 0.000, B 0.000, C 0.000 }
gfCNCPoint2[16042] = {X 140.4836, Y 30.3963, Z -3.0000, A 0.000, B 0.000, C 0.000 }
gfCNCPoint2[16043] = {X 140.4836, Y 19.6371, Z -3.0000, A 0.000, B 0.000, C 0.000 }
gfCNCPoint2[16044] = {X 137.2909, Y 19.6362, Z -3.0000, A 0.000, B 0.000, C 0.000 }
gfCNCPoint2[16045] = {X 137.2218, Y 19.7475, Z -3.0000, A 0.000, B 0.000, C 0.000 }
gfCNCPoint2[16046] = {X 136.5756, Y 20.4907, Z -3.0000, A 0.000, B 0.000, C 0.000 }
gfCNCPoint2[16047] = {X 135.7702, Y 21.0573, Z -3.0000, A 0.000, B 0.000, C 0.000 }
gfCNCPoint2[16048] = {X 134.8524, Y 21.4145, Z -3.0000, A 0.000, B 0.000, C 0.000 }
gfCNCPoint2[16049] = {X 133.8758, Y 21.5414, Z -3.0000, A 0.000, B 0.000, C 0.000 }
gfCNCPoint2[16050] = {X 133.2006, Y 21.5415, Z -3.0000, A 0.000, B 0.000, C 0.000 }
gfCNCPoint2[16051] = {X 132.2928, Y 21.4392, Z -3.0000, A 0.000, B 0.000, C 0.000 }
gfCNCPoint2[16052] = {X 131.4304, Y 21.1375, Z -3.0000, A 0.000, B 0.000, C 0.000 }
gfCNCPoint2[16053] = {X 130.6568, Y 20.6514, Z -3.0000, A 0.000, B 0.000, C 0.000 }
gfCNCPoint2[16054] = {X 130.0108, Y 20.0054, Z -3.0000, A 0.000, B 0.000, C 0.000 }
gfCNCPoint2[16055] = {X 129.5247, Y 19.2318, Z -3.0000, A 0.000, B 0.000, C 0.000 }
gfCNCPoint2[16056] = {X 129.2229, Y 18.3694, Z -3.0000, A 0.000, B 0.000, C 0.000 }
gfCNCPoint2[16057] = {X 129.1206, Y 17.4615, Z -3.0000, A 0.000, B 0.000, C 0.000 }
gfCNCPoint2[16058] = {X 129.1206, Y 10.4835, Z -3.0000, A 0.000, B 0.000, C 0.000 }
gfCNCPoint2[16059] = {X 129.2215, Y 9.5820, Z -3.0000, A 0.000, B 0.000, C 0.000 }
gfCNCPoint2[16060] = {X 129.5191, Y 8.7250, Z -3.0000, A 0.000, B 0.000, C 0.000 }
gfCNCPoint2[16061] = {X 129.9986, Y 7.9550, Z -3.0000, A 0.000, B 0.000, C 0.000 }
gfCNCPoint2[16062] = {X 130.6365, Y 7.3099, Z -3.0000, A 0.000, B 0.000, C 0.000 }
gfCNCPoint2[16063] = {X 131.4011, Y 6.8218, Z -3.0000, A 0.000, B 0.000, C 0.000 }
gfCNCPoint2[16064] = {X 132.2547, Y 6.5147, Z -3.0000, A 0.000, B 0.000, C 0.000 }
gfCNCPoint2[16065] = {X 133.1551, Y 6.4038, Z -3.0000, A 0.000, B 0.000, C 0.000 }
gfCNCPoint2[16066] = {X 133.8841, Y 6.4037, Z -3.0000, A 0.000, B 0.000, C 0.000 }
gfCNCPoint2[16067] = {X 134.6875, Y 6.4920, Z -3.0000, A 0.000, B 0.000, C 0.000 }
gfCNCPoint2[16068] = {X 135.4577, Y 6.7369, Z -3.0000, A 0.000, B 0.000, C 0.000 }
gfCNCPoint2[16069] = {X 136.1645, Y 7.1288, Z -3.0000, A 0.000, B 0.000, C 0.000 }
gfCNCPoint2[16070] = {X 136.7802, Y 7.6524, Z -3.0000, A 0.000, B 0.000, C 0.000 }
gfCNCPoint2[16071] = {X 137.2806, Y 8.2870, Z -3.0000, A 0.000, B 0.000, C 0.000 }
gfCNCPoint2[16072] = {X 155.2414, Y 8.2882, Z -3.0000, A 0.000, B 0.000, C 0.000 }
gfCNCPoint2[16073] = {X 155.2868, Y 8.2186, Z -3.0000, A 0.000, B 0.000, C 0.000 }
gfCNCPoint2[16074] = {X 155.3336, Y 8.1500, Z -3.0000, A 0.000, B 0.000, C 0.000 }
gfCNCPoint2[16075] = {X 155.9787, Y 7.4262, Z -3.0000, A 0.000, B 0.000, C 0.000 }
gfCNCPoint2[16076] = {X 156.7765, Y 6.8750, Z -3.0000, A 0.000, B 0.000, C 0.000 }
gfCNCPoint2[16077] = {X 157.6817, Y 6.5276, Z -3.0000, A 0.000, B 0.000, C 0.000 }
gfCNCPoint2[16078] = {X 158.6434, Y 6.4037, Z -3.0000, A 0.000, B 0.000, C 0.000 }
gfCNCPoint2[16079] = {X 159.3750, Y 6.4039, Z -3.0000, A 0.000, B 0.000, C 0.000 }
gfCNCPoint2[16080] = {X 160.2741, Y 6.5161, Z -3.0000, A 0.000, B 0.000, C 0.000 }
gfCNCPoint2[16081] = {X 161.1263, Y 6.8241, Z -3.0000, A 0.000, B 0.000, C 0.000 }
gfCNCPoint2[16082] = {X 161.8895, Y 7.3126, Z -3.0000, A 0.000, B 0.000, C 0.000 }
gfCNCPoint2[16083] = {X 162.5260, Y 7.9574, Z -3.0000, A 0.000, B 0.000, C 0.000 }
gfCNCPoint2[16084] = {X 163.0046, Y 8.7269, Z -3.0000, A 0.000, B 0.000, C 0.000 }
gfCNCPoint2[16085] = {X 163.3015, Y 9.5830, Z -3.0000, A 0.000, B 0.000, C 0.000 }
gfCNCPoint2[16086] = {X 163.4021, Y 10.4835, Z -3.0000, A 0.000, B 0.000, C 0.000 }
gfCNCPoint2[16087] = {X 163.4021, Y 17.4615, Z -3.0000, A 0.000, B 0.000, C 0.000 }
gfCNCPoint2[16088] = {X 163.3015, Y 18.3621, Z -3.0000, A 0.000, B 0.000, C 0.000 }
gfCNCPoint2[16089] = {X 163.0046, Y 19.2182, Z -3.0000, A 0.000, B 0.000, C 0.000 }
gfCNCPoint2[16090] = {X 162.5260, Y 19.9876, Z -3.0000, A 0.000, B 0.000, C 0.000 }
gfCNCPoint2[16091] = {X 161.8895, Y 20.6325, Z -3.0000, A 0.000, B 0.000, C 0.000 }
gfCNCPoint2[16092] = {X 161.1263, Y 21.1209, Z -3.0000, A 0.000, B 0.000, C 0.000 }
gfCNCPoint2[16093] = {X 160.2741, Y 21.4289, Z -3.0000, A 0.000, B 0.000, C 0.000 }
gfCNCPoint2[16094] = {X 159.3750, Y 21.5412, Z -3.0000, A 0.000, B 0.000, C 0.000 }
gfCNCPoint2[16095] = {X 158.6802, Y 21.5415, Z -3.0000, A 0.000, B 0.000, C 0.000 }
gfCNCPoint2[16096] = {X 157.8634, Y 21.4558, Z -3.0000, A 0.000, B 0.000, C 0.000 }
gfCNCPoint2[16097] = {X 157.0799, Y 21.2097, Z -3.0000, A 0.000, B 0.000, C 0.000 }
gfCNCPoint2[16098] = {X 156.3608, Y 20.8130, Z -3.0000, A 0.000, B 0.000, C 0.000 }
gfCNCPoint2[16099] = {X 155.7348, Y 20.2814, Z -3.0000, A 0.000, B 0.000, C 0.000 }
gfCNCPoint2[16100] = {X 155.2267, Y 19.6362, Z -3.0000, A 0.000, B 0.000, C 0.000 }
gfCNCPoint2[16101] = {X 152.0360, Y 19.6377, Z -3.0000, A 0.000, B 0.000, C 0.000 }
gfCNCPoint2[16102] = {X 152.0344, Y 40.9684, Z -3.0000, A 0.000, B 0.000, C 0.000 }
gfCNCPoint2[16103] = {X 152.5609, Y 41.5352, Z -3.0000, A 0.000, B 0.000, C 0.000 }
gfCNCPoint2[16104] = {X 152.6499, Y 41.6414, Z -3.0000, A 0.000, B 0.000, C 0.000 }
gfCNCPoint2[16105] = {X 153.1457, Y 42.4208, Z -3.0000, A 0.000, B 0.000, C 0.000 }
gfCNCPoint2[16106] = {X 153.4552, Y 43.2911, Z -3.0000, A 0.000, B 0.000, C 0.000 }
gfCNCPoint2[16107] = {X 153.5631, Y 44.2085, Z -3.0000, A 0.000, B 0.000, C 0.000 }
gfCNCPoint2[16108] = {X 153.5629, Y 45.0392, Z -3.0000, A 0.000, B 0.000, C 0.000 }
gfCNCPoint2[16109] = {X 153.4532, Y 45.9406, Z -3.0000, A 0.000, B 0.000, C 0.000 }
gfCNCPoint2[16110] = {X 153.1468, Y 46.7954, Z -3.0000, A 0.000, B 0.000, C 0.000 }
gfCNCPoint2[16111] = {X 152.6589, Y 47.5613, Z -3.0000, A 0.000, B 0.000, C 0.000 }
gfCNCPoint2[16112] = {X 152.0138, Y 48.2003, Z -3.0000, A 0.000, B 0.000, C 0.000 }
gfCNCPoint2[16113] = {X 151.2432, Y 48.6808, Z -3.0000, A 0.000, B 0.000, C 0.000 }
gfCNCPoint2[16114] = {X 150.3855, Y 48.9789, Z -3.0000, A 0.000, B 0.000, C 0.000 }
gfCNCPoint2[16115] = {X 149.4831, Y 49.0800, Z -3.0000, A 0.000, B 0.000, C 0.000 }
gfCNCPoint2[16116] = {X 143.0396, Y 49.0800, Z -3.0000, A 0.000, B 0.000, C 0.000 }
gfCNCPoint2[16117] = {X 142.1362, Y 48.9787, Z -3.0000, A 0.000, B 0.000, C 0.000 }
gfCNCPoint2[16118] = {X 141.2777, Y 48.6799, Z -3.0000, A 0.000, B 0.000, C 0.000 }
gfCNCPoint2[16119] = {X 140.5066, Y 48.1985, Z -3.0000, A 0.000, B 0.000, C 0.000 }
gfCNCPoint2[16120] = {X 139.8613, Y 47.5582, Z -3.0000, A 0.000, B 0.000, C 0.000 }
gfCNCPoint2[16121] = {X 139.3737, Y 46.7910, Z -3.0000, A 0.000, B 0.000, C 0.000 }
gfCNCPoint2[16122] = {X 139.0682, Y 45.9349, Z -3.0000, A 0.000, B 0.000, C 0.000 }
gfCNCPoint2[16123] = {X 138.9598, Y 45.0323, Z -3.0000, A 0.000, B 0.000, C 0.000 }
gfCNCPoint2[16124] = {X 138.9600, Y 44.1527, Z -3.0000, A 0.000, B 0.000, C 0.000 }
gfCNCPoint2[16125] = {X 139.0706, Y 43.2637, Z -3.0000, A 0.000, B 0.000, C 0.000 }
gfCNCPoint2[16126] = {X 139.3725, Y 42.4203, Z -3.0000, A 0.000, B 0.000, C 0.000 }
gfCNCPoint2[16127] = {X 139.8512, Y 41.6631, Z -3.0000, A 0.000, B 0.000, C 0.000 }
gfCNCPoint2[16128] = {X 140.4836, Y 41.0287, Z -3.0000, A 0.000, B 0.000, C 0.000 }
gfCNCPoint2[16129] = {X 140.4836, Y 30.3963, Z -3.0000, A 0.000, B 0.000, C 0.000 }
gfCNCPoint2[16130] = {X 136.4836, Y 30.3963, Z -3.0000, A 0.000, B 0.000, C 0.000 }
gfCNCPoint2[16131] = {X 140.5636, Y 30.3963, Z -3.0000, A 0.000, B 0.000, C 0.000 }
gfCNCPoint2[16132] = {X 140.5636, Y 19.9570, Z -3.0000, A 0.000, B 0.000, C 0.000 }
gfCNCPoint2[16133] = {X 140.5647, Y 19.5571, Z -3.0000, A 0.000, B 0.000, C 0.000 }
gfCNCPoint2[16134] = {X 137.2663, Y 19.5562, Z -3.0000, A 0.000, B 0.000, C 0.000 }
gfCNCPoint2[16135] = {X 137.2438, Y 19.5603, Z -3.0000, A 0.000, B 0.000, C 0.000 }
gfCNCPoint2[16136] = {X 137.1372, Y 19.7295, Z -3.0000, A 0.000, B 0.000, C 0.000 }
gfCNCPoint2[16137] = {X 136.4977, Y 20.4530, Z -3.0000, A 0.000, B 0.000, C 0.000 }
gfCNCPoint2[16138] = {X 135.7035, Y 21.0022, Z -3.0000, A 0.000, B 0.000, C 0.000 }
gfCNCPoint2[16139] = {X 134.8007, Y 21.3450, Z -3.0000, A 0.000, B 0.000, C 0.000 }
gfCNCPoint2[16140] = {X 133.8421, Y 21.4615, Z -3.0000, A 0.000, B 0.000, C 0.000 }
gfCNCPoint2[16141] = {X 133.2006, Y 21.4615, Z -3.0000, A 0.000, B 0.000, C 0.000 }
gfCNCPoint2[16142] = {X 132.3106, Y 21.3613, Z -3.0000, A 0.000, B 0.000, C 0.000 }
gfCNCPoint2[16143] = {X 131.4651, Y 21.0654, Z -3.0000, A 0.000, B 0.000, C 0.000 }
gfCNCPoint2[16144] = {X 130.7067, Y 20.5889, Z -3.0000, A 0.000, B 0.000, C 0.000 }
gfCNCPoint2[16145] = {X 130.0733, Y 19.9555, Z -3.0000, A 0.000, B 0.000, C 0.000 }
gfCNCPoint2[16146] = {X 129.5968, Y 19.1971, Z -3.0000, A 0.000, B 0.000, C 0.000 }
gfCNCPoint2[16147] = {X 129.3009, Y 18.3516, Z -3.0000, A 0.000, B 0.000, C 0.000 }
gfCNCPoint2[16148] = {X 129.2006, Y 17.4615, Z -3.0000, A 0.000, B 0.000, C 0.000 }
gfCNCPoint2[16149] = {X 129.2006, Y 10.4835, Z -3.0000, A 0.000, B 0.000, C 0.000 }
gfCNCPoint2[16150] = {X 129.3009, Y 9.5934, Z -3.0000, A 0.000, B 0.000, C 0.000 }
gfCNCPoint2[16151] = {X 129.5968, Y 8.7480, Z -3.0000, A 0.000, B 0.000, C 0.000 }
gfCNCPoint2[16152] = {X 130.0733, Y 7.9895, Z -3.0000, A 0.000, B 0.000, C 0.000 }
gfCNCPoint2[16153] = {X 130.7067, Y 7.3562, Z -3.0000, A 0.000, B 0.000, C 0.000 }
gfCNCPoint2[16154] = {X 131.4651, Y 6.8796, Z -3.0000, A 0.000, B 0.000, C 0.000 }
gfCNCPoint2[16155] = {X 132.3106, Y 6.5838, Z -3.0000, A 0.000, B 0.000, C 0.000 }
gfCNCPoint2[16156] = {X 133.2007, Y 6.4835, Z -3.0000, A 0.000, B 0.000, C 0.000 }
gfCNCPoint2[16157] = {X 133.8833, Y 6.4837, Z -3.0000, A 0.000, B 0.000, C 0.000 }
gfCNCPoint2[16158] = {X 134.6795, Y 6.5721, Z -3.0000, A 0.000, B 0.000, C 0.000 }
gfCNCPoint2[16159] = {X 135.4420, Y 6.8173, Z -3.0000, A 0.000, B 0.000, C 0.000 }
gfCNCPoint2[16160] = {X 136.1405, Y 7.2096, Z -3.0000, A 0.000, B 0.000, C 0.000 }
gfCNCPoint2[16161] = {X 136.7467, Y 7.7332, Z -3.0000, A 0.000, B 0.000, C 0.000 }
gfCNCPoint2[16162] = {X 137.2365, Y 8.3670, Z -3.0000, A 0.000, B 0.000, C 0.000 }
gfCNCPoint2[16163] = {X 155.2276, Y 8.3670, Z -3.0000, A 0.000, B 0.000, C 0.000 }
gfCNCPoint2[16164] = {X 155.2814, Y 8.3748, Z -3.0000, A 0.000, B 0.000, C 0.000 }
gfCNCPoint2[16165] = {X 155.3391, Y 8.2845, Z -3.0000, A 0.000, B 0.000, C 0.000 }
gfCNCPoint2[16166] = {X 155.3992, Y 8.1958, Z -3.0000, A 0.000, B 0.000, C 0.000 }
gfCNCPoint2[16167] = {X 156.0385, Y 7.4801, Z -3.0000, A 0.000, B 0.000, C 0.000 }
gfCNCPoint2[16168] = {X 156.8299, Y 6.9373, Z -3.0000, A 0.000, B 0.000, C 0.000 }
gfCNCPoint2[16169] = {X 157.7279, Y 6.5986, Z -3.0000, A 0.000, B 0.000, C 0.000 }
gfCNCPoint2[16170] = {X 158.6806, Y 6.4835, Z -3.0000, A 0.000, B 0.000, C 0.000 }
gfCNCPoint2[16171] = {X 159.3739, Y 6.4839, Z -3.0000, A 0.000, B 0.000, C 0.000 }
gfCNCPoint2[16172] = {X 160.2554, Y 6.5939, Z -3.0000, A 0.000, B 0.000, C 0.000 }
gfCNCPoint2[16173] = {X 161.0909, Y 6.8959, Z -3.0000, A 0.000, B 0.000, C 0.000 }
gfCNCPoint2[16174] = {X 161.8391, Y 7.3747, Z -3.0000, A 0.000, B 0.000, C 0.000 }
gfCNCPoint2[16175] = {X 162.4632, Y 8.0070, Z -3.0000, A 0.000, B 0.000, C 0.000 }
gfCNCPoint2[16176] = {X 162.9324, Y 8.7613, Z -3.0000, A 0.000, B 0.000, C 0.000 }
gfCNCPoint2[16177] = {X 163.2234, Y 9.6007, Z -3.0000, A 0.000, B 0.000, C 0.000 }
gfCNCPoint2[16178] = {X 163.3221, Y 10.4835, Z -3.0000, A 0.000, B 0.000, C 0.000 }
gfCNCPoint2[16179] = {X 163.3221, Y 17.4615, Z -3.0000, A 0.000, B 0.000, C 0.000 }
gfCNCPoint2[16180] = {X 163.2218, Y 18.3516, Z -3.0000, A 0.000, B 0.000, C 0.000 }
gfCNCPoint2[16181] = {X 162.9260, Y 19.1971, Z -3.0000, A 0.000, B 0.000, C 0.000 }
gfCNCPoint2[16182] = {X 162.4494, Y 19.9555, Z -3.0000, A 0.000, B 0.000, C 0.000 }
gfCNCPoint2[16183] = {X 161.8160, Y 20.5889, Z -3.0000, A 0.000, B 0.000, C 0.000 }
gfCNCPoint2[16184] = {X 161.0576, Y 21.0654, Z -3.0000, A 0.000, B 0.000, C 0.000 }
gfCNCPoint2[16185] = {X 160.2121, Y 21.3613, Z -3.0000, A 0.000, B 0.000, C 0.000 }
gfCNCPoint2[16186] = {X 159.3221, Y 21.4615, Z -3.0000, A 0.000, B 0.000, C 0.000 }
gfCNCPoint2[16187] = {X 158.6806, Y 21.4615, Z -3.0000, A 0.000, B 0.000, C 0.000 }
gfCNCPoint2[16188] = {X 157.8711, Y 21.3757, Z -3.0000, A 0.000, B 0.000, C 0.000 }
gfCNCPoint2[16189] = {X 157.0953, Y 21.1292, Z -3.0000, A 0.000, B 0.000, C 0.000 }
gfCNCPoint2[16190] = {X 156.3847, Y 20.7322, Z -3.0000, A 0.000, B 0.000, C 0.000 }
gfCNCPoint2[16191] = {X 155.7682, Y 20.2006, Z -3.0000, A 0.000, B 0.000, C 0.000 }
gfCNCPoint2[16192] = {X 155.2709, Y 19.5562, Z -3.0000, A 0.000, B 0.000, C 0.000 }
gfCNCPoint2[16193] = {X 151.9560, Y 19.5578, Z -3.0000, A 0.000, B 0.000, C 0.000 }
gfCNCPoint2[16194] = {X 151.9544, Y 40.9999, Z -3.0000, A 0.000, B 0.000, C 0.000 }
gfCNCPoint2[16195] = {X 152.5009, Y 41.5881, Z -3.0000, A 0.000, B 0.000, C 0.000 }
gfCNCPoint2[16196] = {X 152.5881, Y 41.6922, Z -3.0000, A 0.000, B 0.000, C 0.000 }
gfCNCPoint2[16197] = {X 153.0740, Y 42.4563, Z -3.0000, A 0.000, B 0.000, C 0.000 }
gfCNCPoint2[16198] = {X 153.3774, Y 43.3095, Z -3.0000, A 0.000, B 0.000, C 0.000 }
gfCNCPoint2[16199] = {X 153.4831, Y 44.2089, Z -3.0000, A 0.000, B 0.000, C 0.000 }
gfCNCPoint2[16200] = {X 153.4829, Y 45.0384, Z -3.0000, A 0.000, B 0.000, C 0.000 }
gfCNCPoint2[16201] = {X 153.3753, Y 45.9222, Z -3.0000, A 0.000, B 0.000, C 0.000 }
gfCNCPoint2[16202] = {X 153.0750, Y 46.7602, Z -3.0000, A 0.000, B 0.000, C 0.000 }
gfCNCPoint2[16203] = {X 152.5967, Y 47.5111, Z -3.0000, A 0.000, B 0.000, C 0.000 }
gfCNCPoint2[16204] = {X 151.9642, Y 48.1376, Z -3.0000, A 0.000, B 0.000, C 0.000 }
gfCNCPoint2[16205] = {X 151.2087, Y 48.6086, Z -3.0000, A 0.000, B 0.000, C 0.000 }
gfCNCPoint2[16206] = {X 150.3678, Y 48.9009, Z -3.0000, A 0.000, B 0.000, C 0.000 }
gfCNCPoint2[16207] = {X 149.4831, Y 49.0000, Z -3.0000, A 0.000, B 0.000, C 0.000 }
gfCNCPoint2[16208] = {X 143.0396, Y 49.0000, Z -3.0000, A 0.000, B 0.000, C 0.000 }
gfCNCPoint2[16209] = {X 142.1495, Y 48.8997, Z -3.0000, A 0.000, B 0.000, C 0.000 }
gfCNCPoint2[16210] = {X 141.3041, Y 48.6039, Z -3.0000, A 0.000, B 0.000, C 0.000 }
gfCNCPoint2[16211] = {X 140.5457, Y 48.1273, Z -3.0000, A 0.000, B 0.000, C 0.000 }
gfCNCPoint2[16212] = {X 139.9123, Y 47.4939, Z -3.0000, A 0.000, B 0.000, C 0.000 }
gfCNCPoint2[16213] = {X 139.4357, Y 46.7355, Z -3.0000, A 0.000, B 0.000, C 0.000 }
gfCNCPoint2[16214] = {X 139.1399, Y 45.8900, Z -3.0000, A 0.000, B 0.000, C 0.000 }
gfCNCPoint2[16215] = {X 139.0396, Y 45.0000, Z -3.0000, A 0.000, B 0.000, C 0.000 }
gfCNCPoint2[16216] = {X 139.0400, Y 44.1538, Z -3.0000, A 0.000, B 0.000, C 0.000 }
gfCNCPoint2[16217] = {X 139.1506, Y 43.2730, Z -3.0000, A 0.000, B 0.000, C 0.000 }
gfCNCPoint2[16218] = {X 139.4528, Y 42.4382, Z -3.0000, A 0.000, B 0.000, C 0.000 }
gfCNCPoint2[16219] = {X 139.9317, Y 41.6907, Z -3.0000, A 0.000, B 0.000, C 0.000 }
gfCNCPoint2[16220] = {X 140.5636, Y 41.0672, Z -3.0000, A 0.000, B 0.000, C 0.000 }
gfCNCPoint2[16221] = {X 140.5636, Y 30.3963, Z -3.0000, A 0.000, B 0.000, C 0.000 }
gfCNCPoint2[16222] = {X 136.4836, Y 30.3963, Z -3.0000, A 0.000, B 0.000, C 0.000 }
gfCNCPoint2[16223] = {X 136.4836, Y 30.3963, Z 0.0000, A 0.000, B 0.000, C 0.000 }
gfCNCPoint2[16224] = {X 136.4836, Y 30.3963, Z 11.0000, A 0.000, B 0.000, C 0.000 }
gfCNCPoint2[16225] = {X 137.6637, Y 74.8932, Z 11.0000, A 0.000, B 0.000, C 0.000 }
gfCNCPoint2[16226] = {X 137.6637, Y 74.8932, Z 0.0000, A 0.000, B 0.000, C 0.000 }
gfCNCPoint2[16227] = {X 137.6637, Y 74.8932, Z -3.0000, A 0.000, B 0.000, C 0.000 }
gfCNCPoint2[16228] = {X 140.6804, Y 77.6403, Z -3.0000, A 0.000, B 0.000, C 0.000 }
gfCNCPoint2[16229] = {X 155.6327, Y 61.2206, Z -3.0000, A 0.000, B 0.000, C 0.000 }
gfCNCPoint2[16230] = {X 155.2775, Y 60.5147, Z -3.0000, A 0.000, B 0.000, C 0.000 }
gfCNCPoint2[16231] = {X 155.0569, Y 59.7560, Z -3.0000, A 0.000, B 0.000, C 0.000 }
gfCNCPoint2[16232] = {X 154.9781, Y 58.9697, Z -3.0000, A 0.000, B 0.000, C 0.000 }
gfCNCPoint2[16233] = {X 154.9780, Y 58.0000, Z -3.0000, A 0.000, B 0.000, C 0.000 }
gfCNCPoint2[16234] = {X 155.0863, Y 57.0387, Z -3.0000, A 0.000, B 0.000, C 0.000 }
gfCNCPoint2[16235] = {X 155.4058, Y 56.1256, Z -3.0000, A 0.000, B 0.000, C 0.000 }
gfCNCPoint2[16236] = {X 155.9204, Y 55.3065, Z -3.0000, A 0.000, B 0.000, C 0.000 }
gfCNCPoint2[16237] = {X 156.6045, Y 54.6225, Z -3.0000, A 0.000, B 0.000, C 0.000 }
gfCNCPoint2[16238] = {X 157.4236, Y 54.1078, Z -3.0000, A 0.000, B 0.000, C 0.000 }
gfCNCPoint2[16239] = {X 158.3367, Y 53.7883, Z -3.0000, A 0.000, B 0.000, C 0.000 }
gfCNCPoint2[16240] = {X 159.2980, Y 53.6800, Z -3.0000, A 0.000, B 0.000, C 0.000 }
gfCNCPoint2[16241] = {X 178.5335, Y 53.6800, Z -3.0000, A 0.000, B 0.000, C 0.000 }
gfCNCPoint2[16242] = {X 179.4948, Y 53.7883, Z -3.0000, A 0.000, B 0.000, C 0.000 }
gfCNCPoint2[16243] = {X 180.4079, Y 54.1078, Z -3.0000, A 0.000, B 0.000, C 0.000 }
gfCNCPoint2[16244] = {X 181.2270, Y 54.6225, Z -3.0000, A 0.000, B 0.000, C 0.000 }
gfCNCPoint2[16245] = {X 181.9110, Y 55.3065, Z -3.0000, A 0.000, B 0.000, C 0.000 }
gfCNCPoint2[16246] = {X 182.4257, Y 56.1256, Z -3.0000, A 0.000, B 0.000, C 0.000 }
gfCNCPoint2[16247] = {X 182.7452, Y 57.0387, Z -3.0000, A 0.000, B 0.000, C 0.000 }
gfCNCPoint2[16248] = {X 182.8535, Y 58.0000, Z -3.0000, A 0.000, B 0.000, C 0.000 }
gfCNCPoint2[16249] = {X 182.8535, Y 58.9342, Z -3.0000, A 0.000, B 0.000, C 0.000 }
gfCNCPoint2[16250] = {X 182.7808, Y 59.7235, Z -3.0000, A 0.000, B 0.000, C 0.000 }
gfCNCPoint2[16251] = {X 182.5651, Y 60.4861, Z -3.0000, A 0.000, B 0.000, C 0.000 }
gfCNCPoint2[16252] = {X 182.2137, Y 61.1966, Z -3.0000, A 0.000, B 0.000, C 0.000 }
gfCNCPoint2[16253] = {X 209.4780, Y 90.9540, Z -3.0000, A 0.000, B 0.000, C 0.000 }
gfCNCPoint2[16254] = {X 210.1357, Y 91.6214, Z -3.0000, A 0.000, B 0.000, C 0.000 }
gfCNCPoint2[16255] = {X 210.8404, Y 92.2391, Z -3.0000, A 0.000, B 0.000, C 0.000 }
gfCNCPoint2[16256] = {X 211.1141, Y 92.4123, Z -3.0000, A 0.000, B 0.000, C 0.000 }
gfCNCPoint2[16257] = {X 211.4210, Y 92.5159, Z -3.0000, A 0.000, B 0.000, C 0.000 }
gfCNCPoint2[16258] = {X 213.4039, Y 92.8252, Z -3.0000, A 0.000, B 0.000, C 0.000 }
gfCNCPoint2[16259] = {X 214.4545, Y 92.7364, Z -3.0000, A 0.000, B 0.000, C 0.000 }
gfCNCPoint2[16260] = {X 215.5072, Y 92.6762, Z -3.0000, A 0.000, B 0.000, C 0.000 }
gfCNCPoint2[16261] = {X 216.1773, Y 92.6030, Z -3.0000, A 0.000, B 0.000, C 0.000 }
gfCNCPoint2[16262] = {X 216.8225, Y 92.4079, Z -3.0000, A 0.000, B 0.000, C 0.000 }
gfCNCPoint2[16263] = {X 217.4209, Y 92.0978, Z -3.0000, A 0.000, B 0.000, C 0.000 }
gfCNCPoint2[16264] = {X 222.9613, Y 88.5223, Z -3.0000, A 0.000, B 0.000, C 0.000 }
gfCNCPoint2[16265] = {X 245.8288, Y 73.8995, Z -3.0000, A 0.000, B 0.000, C 0.000 }
gfCNCPoint2[16266] = {X 221.6305, Y 64.4031, Z -3.0000, A 0.000, B 0.000, C 0.000 }
gfCNCPoint2[16267] = {X 219.8632, Y 63.8116, Z -3.0000, A 0.000, B 0.000, C 0.000 }
gfCNCPoint2[16268] = {X 218.0398, Y 63.4260, Z -3.0000, A 0.000, B 0.000, C 0.000 }
gfCNCPoint2[16269] = {X 216.1842, Y 63.2516, Z -3.0000, A 0.000, B 0.000, C 0.000 }
gfCNCPoint2[16270] = {X 215.2524, Y 63.1173, Z -3.0000, A 0.000, B 0.000, C 0.000 }
gfCNCPoint2[16271] = {X 214.3717, Y 62.7843, Z -3.0000, A 0.000, B 0.000, C 0.000 }
gfCNCPoint2[16272] = {X 213.5841, Y 62.2685, Z -3.0000, A 0.000, B 0.000, C 0.000 }
gfCNCPoint2[16273] = {X 212.9270, Y 61.5942, Z -3.0000, A 0.000, B 0.000, C 0.000 }
gfCNCPoint2[16274] = {X 212.4315, Y 60.7936, Z -3.0000, A 0.000, B 0.000, C 0.000 }
gfCNCPoint2[16275] = {X 212.1213, Y 59.9047, Z -3.0000, A 0.000, B 0.000, C 0.000 }
gfCNCPoint2[16276] = {X 212.0110, Y 58.9697, Z -3.0000, A 0.000, B 0.000, C 0.000 }
gfCNCPoint2[16277] = {X 212.0108, Y 58.0000, Z -3.0000, A 0.000, B 0.000, C 0.000 }
gfCNCPoint2[16278] = {X 212.1191, Y 57.0387, Z -3.0000, A 0.000, B 0.000, C 0.000 }
gfCNCPoint2[16279] = {X 212.4386, Y 56.1256, Z -3.0000, A 0.000, B 0.000, C 0.000 }
gfCNCPoint2[16280] = {X 212.9533, Y 55.3065, Z -3.0000, A 0.000, B 0.000, C 0.000 }
gfCNCPoint2[16281] = {X 213.6373, Y 54.6225, Z -3.0000, A 0.000, B 0.000, C 0.000 }
gfCNCPoint2[16282] = {X 214.4564, Y 54.1078, Z -3.0000, A 0.000, B 0.000, C 0.000 }
gfCNCPoint2[16283] = {X 215.3695, Y 53.7883, Z -3.0000, A 0.000, B 0.000, C 0.000 }
gfCNCPoint2[16284] = {X 216.3308, Y 53.6800, Z -3.0000, A 0.000, B 0.000, C 0.000 }
gfCNCPoint2[16285] = {X 237.2617, Y 53.6800, Z -3.0000, A 0.000, B 0.000, C 0.000 }
gfCNCPoint2[16286] = {X 238.2230, Y 53.7883, Z -3.0000, A 0.000, B 0.000, C 0.000 }
gfCNCPoint2[16287] = {X 239.1361, Y 54.1078, Z -3.0000, A 0.000, B 0.000, C 0.000 }
gfCNCPoint2[16288] = {X 239.9552, Y 54.6225, Z -3.0000, A 0.000, B 0.000, C 0.000 }
gfCNCPoint2[16289] = {X 240.6392, Y 55.3065, Z -3.0000, A 0.000, B 0.000, C 0.000 }
gfCNCPoint2[16290] = {X 241.1539, Y 56.1256, Z -3.0000, A 0.000, B 0.000, C 0.000 }
gfCNCPoint2[16291] = {X 241.4734, Y 57.0387, Z -3.0000, A 0.000, B 0.000, C 0.000 }
gfCNCPoint2[16292] = {X 241.5817, Y 58.0000, Z -3.0000, A 0.000, B 0.000, C 0.000 }
gfCNCPoint2[16293] = {X 241.5817, Y 58.2327, Z -3.0000, A 0.000, B 0.000, C 0.000 }
gfCNCPoint2[16294] = {X 247.4883, Y 60.5353, Z -3.0000, A 0.000, B 0.000, C 0.000 }
gfCNCPoint2[16295] = {X 275.6335, Y 71.7027, Z -3.0000, A 0.000, B 0.000, C 0.000 }
gfCNCPoint2[16296] = {X 275.6343, Y 63.2124, Z -3.0000, A 0.000, B 0.000, C 0.000 }
gfCNCPoint2[16297] = {X 274.7825, Y 63.0034, Z -3.0000, A 0.000, B 0.000, C 0.000 }
gfCNCPoint2[16298] = {X 273.9905, Y 62.6266, Z -3.0000, A 0.000, B 0.000, C 0.000 }
gfCNCPoint2[16299] = {X 273.2910, Y 62.0977, Z -3.0000, A 0.000, B 0.000, C 0.000 }
gfCNCPoint2[16300] = {X 272.7126, Y 61.4384, Z -3.0000, A 0.000, B 0.000, C 0.000 }
gfCNCPoint2[16301] = {X 272.2794, Y 60.6758, Z -3.0000, A 0.000, B 0.000, C 0.000 }
gfCNCPoint2[16302] = {X 272.0091, Y 59.8415, Z -3.0000, A 0.000, B 0.000, C 0.000 }
gfCNCPoint2[16303] = {X 271.9128, Y 58.9697, Z -3.0000, A 0.000, B 0.000, C 0.000 }
gfCNCPoint2[16304] = {X 271.9127, Y 58.0000, Z -3.0000, A 0.000, B 0.000, C 0.000 }
gfCNCPoint2[16305] = {X 272.0210, Y 57.0387, Z -3.0000, A 0.000, B 0.000, C 0.000 }
gfCNCPoint2[16306] = {X 272.3405, Y 56.1256, Z -3.0000, A 0.000, B 0.000, C 0.000 }
gfCNCPoint2[16307] = {X 272.8552, Y 55.3065, Z -3.0000, A 0.000, B 0.000, C 0.000 }
gfCNCPoint2[16308] = {X 273.5392, Y 54.6225, Z -3.0000, A 0.000, B 0.000, C 0.000 }
gfCNCPoint2[16309] = {X 274.3583, Y 54.1078, Z -3.0000, A 0.000, B 0.000, C 0.000 }
gfCNCPoint2[16310] = {X 275.2714, Y 53.7883, Z -3.0000, A 0.000, B 0.000, C 0.000 }
gfCNCPoint2[16311] = {X 276.2327, Y 53.6800, Z -3.0000, A 0.000, B 0.000, C 0.000 }
gfCNCPoint2[16312] = {X 292.7731, Y 53.6800, Z -3.0000, A 0.000, B 0.000, C 0.000 }
gfCNCPoint2[16313] = {X 293.7344, Y 53.7883, Z -3.0000, A 0.000, B 0.000, C 0.000 }
gfCNCPoint2[16314] = {X 294.6475, Y 54.1078, Z -3.0000, A 0.000, B 0.000, C 0.000 }
gfCNCPoint2[16315] = {X 295.4666, Y 54.6225, Z -3.0000, A 0.000, B 0.000, C 0.000 }
gfCNCPoint2[16316] = {X 296.1506, Y 55.3065, Z -3.0000, A 0.000, B 0.000, C 0.000 }
gfCNCPoint2[16317] = {X 296.6653, Y 56.1256, Z -3.0000, A 0.000, B 0.000, C 0.000 }
gfCNCPoint2[16318] = {X 296.9848, Y 57.0387, Z -3.0000, A 0.000, B 0.000, C 0.000 }
gfCNCPoint2[16319] = {X 297.0931, Y 58.0000, Z -3.0000, A 0.000, B 0.000, C 0.000 }
gfCNCPoint2[16320] = {X 297.0931, Y 58.9352, Z -3.0000, A 0.000, B 0.000, C 0.000 }
gfCNCPoint2[16321] = {X 297.0006, Y 59.8116, Z -3.0000, A 0.000, B 0.000, C 0.000 }
gfCNCPoint2[16322] = {X 296.7328, Y 60.6513, Z -3.0000, A 0.000, B 0.000, C 0.000 }
gfCNCPoint2[16323] = {X 296.3009, Y 61.4194, Z -3.0000, A 0.000, B 0.000, C 0.000 }
gfCNCPoint2[16324] = {X 295.7225, Y 62.0844, Z -3.0000, A 0.000, B 0.000, C 0.000 }
gfCNCPoint2[16325] = {X 295.0217, Y 62.6188, Z -3.0000, A 0.000, B 0.000, C 0.000 }
gfCNCPoint2[16326] = {X 294.2273, Y 63.0004, Z -3.0000, A 0.000, B 0.000, C 0.000 }
gfCNCPoint2[16327] = {X 293.3721, Y 63.2135, Z -3.0000, A 0.000, B 0.000, C 0.000 }
gfCNCPoint2[16328] = {X 293.3842, Y 92.7818, Z -3.0000, A 0.000, B 0.000, C 0.000 }
gfCNCPoint2[16329] = {X 294.2367, Y 92.9992, Z -3.0000, A 0.000, B 0.000, C 0.000 }
gfCNCPoint2[16330] = {X 295.0280, Y 93.3836, Z -3.0000, A 0.000, B 0.000, C 0.000 }
gfCNCPoint2[16331] = {X 295.7259, Y 93.9192, Z -3.0000, A 0.000, B 0.000, C 0.000 }
gfCNCPoint2[16332] = {X 296.3019, Y 94.5843, Z -3.0000, A 0.000, B 0.000, C 0.000 }
gfCNCPoint2[16333] = {X 296.7323, Y 95.3515, Z -3.0000, A 0.000, B 0.000, C 0.000 }
gfCNCPoint2[16334] = {X 296.9997, Y 96.1897, Z -3.0000, A 0.000, B 0.000, C 0.000 }
gfCNCPoint2[16335] = {X 297.0931, Y 97.0645, Z -3.0000, A 0.000, B 0.000, C 0.000 }
gfCNCPoint2[16336] = {X 297.0931, Y 98.0000, Z -3.0000, A 0.000, B 0.000, C 0.000 }
gfCNCPoint2[16337] = {X 296.9848, Y 98.9613, Z -3.0000, A 0.000, B 0.000, C 0.000 }
gfCNCPoint2[16338] = {X 296.6653, Y 99.8744, Z -3.0000, A 0.000, B 0.000, C 0.000 }
gfCNCPoint2[16339] = {X 296.1506, Y 100.6935, Z -3.0000, A 0.000, B 0.000, C 0.000 }
gfCNCPoint2[16340] = {X 295.4666, Y 101.3775, Z -3.0000, A 0.000, B 0.000, C 0.000 }
gfCNCPoint2[16341] = {X 294.6475, Y 101.8922, Z -3.0000, A 0.000, B 0.000, C 0.000 }
gfCNCPoint2[16342] = {X 293.7344, Y 102.2117, Z -3.0000, A 0.000, B 0.000, C 0.000 }
gfCNCPoint2[16343] = {X 292.7731, Y 102.3200, Z -3.0000, A 0.000, B 0.000, C 0.000 }
gfCNCPoint2[16344] = {X 276.2327, Y 102.3200, Z -3.0000, A 0.000, B 0.000, C 0.000 }
gfCNCPoint2[16345] = {X 275.2714, Y 102.2117, Z -3.0000, A 0.000, B 0.000, C 0.000 }
gfCNCPoint2[16346] = {X 274.3583, Y 101.8922, Z -3.0000, A 0.000, B 0.000, C 0.000 }
gfCNCPoint2[16347] = {X 273.5392, Y 101.3775, Z -3.0000, A 0.000, B 0.000, C 0.000 }
gfCNCPoint2[16348] = {X 272.8552, Y 100.6935, Z -3.0000, A 0.000, B 0.000, C 0.000 }
gfCNCPoint2[16349] = {X 272.3405, Y 99.8744, Z -3.0000, A 0.000, B 0.000, C 0.000 }
gfCNCPoint2[16350] = {X 272.0210, Y 98.9613, Z -3.0000, A 0.000, B 0.000, C 0.000 }
gfCNCPoint2[16351] = {X 271.9127, Y 98.0000, Z -3.0000, A 0.000, B 0.000, C 0.000 }
gfCNCPoint2[16352] = {X 271.9127, Y 97.0659, Z -3.0000, A 0.000, B 0.000, C 0.000 }
gfCNCPoint2[16353] = {X 272.0026, Y 96.1891, Z -3.0000, A 0.000, B 0.000, C 0.000 }
gfCNCPoint2[16354] = {X 272.2686, Y 95.3488, Z -3.0000, A 0.000, B 0.000, C 0.000 }
gfCNCPoint2[16355] = {X 272.6996, Y 94.5800, Z -3.0000, A 0.000, B 0.000, C 0.000 }
gfCNCPoint2[16356] = {X 273.2777, Y 93.9147, Z -3.0000, A 0.000, B 0.000, C 0.000 }
gfCNCPoint2[16357] = {X 273.9788, Y 93.3805, Z -3.0000, A 0.000, B 0.000, C 0.000 }
gfCNCPoint2[16358] = {X 274.7737, Y 92.9997, Z -3.0000, A 0.000, B 0.000, C 0.000 }
gfCNCPoint2[16359] = {X 275.6294, Y 92.7883, Z -3.0000, A 0.000, B 0.000, C 0.000 }
gfCNCPoint2[16360] = {X 275.6294, Y 85.5950, Z -3.0000, A 0.000, B 0.000, C 0.000 }
gfCNCPoint2[16361] = {X 262.6396, Y 80.5029, Z -3.0000, A 0.000, B 0.000, C 0.000 }
gfCNCPoint2[16362] = {X 262.2763, Y 80.7316, Z -3.0000, A 0.000, B 0.000, C 0.000 }
gfCNCPoint2[16363] = {X 237.7962, Y 96.5880, Z -3.0000, A 0.000, B 0.000, C 0.000 }
gfCNCPoint2[16364] = {X 237.7998, Y 97.0647, Z -3.0000, A 0.000, B 0.000, C 0.000 }
gfCNCPoint2[16365] = {X 237.7998, Y 98.0000, Z -3.0000, A 0.000, B 0.000, C 0.000 }
gfCNCPoint2[16366] = {X 237.6915, Y 98.9613, Z -3.0000, A 0.000, B 0.000, C 0.000 }
gfCNCPoint2[16367] = {X 237.3720, Y 99.8744, Z -3.0000, A 0.000, B 0.000, C 0.000 }
gfCNCPoint2[16368] = {X 236.8573, Y 100.6935, Z -3.0000, A 0.000, B 0.000, C 0.000 }
gfCNCPoint2[16369] = {X 236.1733, Y 101.3775, Z -3.0000, A 0.000, B 0.000, C 0.000 }
gfCNCPoint2[16370] = {X 235.3542, Y 101.8922, Z -3.0000, A 0.000, B 0.000, C 0.000 }
gfCNCPoint2[16371] = {X 234.4411, Y 102.2117, Z -3.0000, A 0.000, B 0.000, C 0.000 }
gfCNCPoint2[16372] = {X 233.4798, Y 102.3200, Z -3.0000, A 0.000, B 0.000, C 0.000 }
gfCNCPoint2[16373] = {X 214.1790, Y 102.3200, Z -3.0000, A 0.000, B 0.000, C 0.000 }
gfCNCPoint2[16374] = {X 213.7862, Y 102.3021, Z -3.0000, A 0.000, B 0.000, C 0.000 }
gfCNCPoint2[16375] = {X 213.3966, Y 102.2485, Z -3.0000, A 0.000, B 0.000, C 0.000 }
gfCNCPoint2[16376] = {X 213.0070, Y 102.3021, Z -3.0000, A 0.000, B 0.000, C 0.000 }
gfCNCPoint2[16377] = {X 212.6141, Y 102.3200, Z -3.0000, A 0.000, B 0.000, C 0.000 }
gfCNCPoint2[16378] = {X 194.9870, Y 102.3200, Z -3.0000, A 0.000, B 0.000, C 0.000 }
gfCNCPoint2[16379] = {X 194.0257, Y 102.2117, Z -3.0000, A 0.000, B 0.000, C 0.000 }
gfCNCPoint2[16380] = {X 193.1126, Y 101.8922, Z -3.0000, A 0.000, B 0.000, C 0.000 }
gfCNCPoint2[16381] = {X 192.2935, Y 101.3775, Z -3.0000, A 0.000, B 0.000, C 0.000 }
gfCNCPoint2[16382] = {X 191.6094, Y 100.6935, Z -3.0000, A 0.000, B 0.000, C 0.000 }
gfCNCPoint2[16383] = {X 191.0948, Y 99.8744, Z -3.0000, A 0.000, B 0.000, C 0.000 }
gfCNCPoint2[16384] = {X 190.7753, Y 98.9613, Z -3.0000, A 0.000, B 0.000, C 0.000 }
gfCNCPoint2[16385] = {X 190.6670, Y 98.0000, Z -3.0000, A 0.000, B 0.000, C 0.000 }
gfCNCPoint2[16386] = {X 190.6670, Y 97.0659, Z -3.0000, A 0.000, B 0.000, C 0.000 }
gfCNCPoint2[16387] = {X 190.7727, Y 96.1162, Z -3.0000, A 0.000, B 0.000, C 0.000 }
gfCNCPoint2[16388] = {X 191.0846, Y 95.2129, Z -3.0000, A 0.000, B 0.000, C 0.000 }
gfCNCPoint2[16389] = {X 191.5874, Y 94.4003, Z -3.0000, A 0.000, B 0.000, C 0.000 }
gfCNCPoint2[16390] = {X 188.5647, Y 91.1002, Z -3.0000, A 0.000, B 0.000, C 0.000 }
gfCNCPoint2[16391] = {X 150.0898, Y 91.1002, Z -3.0000, A 0.000, B 0.000, C 0.000 }
gfCNCPoint2[16392] = {X 147.1446, Y 94.3631, Z -3.0000, A 0.000, B 0.000, C 0.000 }
gfCNCPoint2[16393] = {X 147.6633, Y 95.1843, Z -3.0000, A 0.000, B 0.000, C 0.000 }
gfCNCPoint2[16394] = {X 147.9869, Y 96.1001, Z -3.0000, A 0.000, B 0.000, C 0.000 }
gfCNCPoint2[16395] = {X 148.0991, Y 97.0649, Z -3.0000, A 0.000, B 0.000, C 0.000 }
gfCNCPoint2[16396] = {X 148.0991, Y 98.0000, Z -3.0000, A 0.000, B 0.000, C 0.000 }
gfCNCPoint2[16397] = {X 147.9908, Y 98.9613, Z -3.0000, A 0.000, B 0.000, C 0.000 }
gfCNCPoint2[16398] = {X 147.6713, Y 99.8744, Z -3.0000, A 0.000, B 0.000, C 0.000 }
gfCNCPoint2[16399] = {X 147.1566, Y 100.6935, Z -3.0000, A 0.000, B 0.000, C 0.000 }
gfCNCPoint2[16400] = {X 146.4726, Y 101.3775, Z -3.0000, A 0.000, B 0.000, C 0.000 }
gfCNCPoint2[16401] = {X 145.6535, Y 101.8922, Z -3.0000, A 0.000, B 0.000, C 0.000 }
gfCNCPoint2[16402] = {X 144.7404, Y 102.2117, Z -3.0000, A 0.000, B 0.000, C 0.000 }
gfCNCPoint2[16403] = {X 143.7791, Y 102.3200, Z -3.0000, A 0.000, B 0.000, C 0.000 }
gfCNCPoint2[16404] = {X 125.0000, Y 102.3200, Z -3.0000, A 0.000, B 0.000, C 0.000 }
gfCNCPoint2[16405] = {X 124.0387, Y 102.2117, Z -3.0000, A 0.000, B 0.000, C 0.000 }
gfCNCPoint2[16406] = {X 123.1256, Y 101.8922, Z -3.0000, A 0.000, B 0.000, C 0.000 }
gfCNCPoint2[16407] = {X 122.3065, Y 101.3775, Z -3.0000, A 0.000, B 0.000, C 0.000 }
gfCNCPoint2[16408] = {X 121.6225, Y 100.6935, Z -3.0000, A 0.000, B 0.000, C 0.000 }
gfCNCPoint2[16409] = {X 121.1078, Y 99.8744, Z -3.0000, A 0.000, B 0.000, C 0.000 }
gfCNCPoint2[16410] = {X 120.7883, Y 98.9613, Z -3.0000, A 0.000, B 0.000, C 0.000 }
gfCNCPoint2[16411] = {X 120.6800, Y 98.0000, Z -3.0000, A 0.000, B 0.000, C 0.000 }
gfCNCPoint2[16412] = {X 120.6800, Y 97.0659, Z -3.0000, A 0.000, B 0.000, C 0.000 }
gfCNCPoint2[16413] = {X 120.7832, Y 96.1271, Z -3.0000, A 0.000, B 0.000, C 0.000 }
gfCNCPoint2[16414] = {X 121.0881, Y 95.2331, Z -3.0000, A 0.000, B 0.000, C 0.000 }
gfCNCPoint2[16415] = {X 121.5799, Y 94.4268, Z -3.0000, A 0.000, B 0.000, C 0.000 }
gfCNCPoint2[16416] = {X 122.2351, Y 93.7466, Z -3.0000, A 0.000, B 0.000, C 0.000 }
gfCNCPoint2[16417] = {X 123.0226, Y 93.2251, Z -3.0000, A 0.000, B 0.000, C 0.000 }
gfCNCPoint2[16418] = {X 123.9046, Y 92.8871, Z -3.0000, A 0.000, B 0.000, C 0.000 }
gfCNCPoint2[16419] = {X 124.8389, Y 92.7489, Z -3.0000, A 0.000, B 0.000, C 0.000 }
gfCNCPoint2[16420] = {X 124.8824, Y 92.7323, Z -3.0000, A 0.000, B 0.000, C 0.000 }
gfCNCPoint2[16421] = {X 124.9279, Y 92.7221, Z -3.0000, A 0.000, B 0.000, C 0.000 }
gfCNCPoint2[16422] = {X 125.4492, Y 92.6448, Z -3.0000, A 0.000, B 0.000, C 0.000 }
gfCNCPoint2[16423] = {X 126.2806, Y 92.5043, Z -3.0000, A 0.000, B 0.000, C 0.000 }
gfCNCPoint2[16424] = {X 127.1006, Y 92.3083, Z -3.0000, A 0.000, B 0.000, C 0.000 }
gfCNCPoint2[16425] = {X 128.3222, Y 91.1565, Z -3.0000, A 0.000, B 0.000, C 0.000 }
gfCNCPoint2[16426] = {X 129.4796, Y 89.9402, Z -3.0000, A 0.000, B 0.000, C 0.000 }
gfCNCPoint2[16427] = {X 140.6804, Y 77.6403, Z -3.0000, A 0.000, B 0.000, C 0.000 }
gfCNCPoint2[16428] = {X 137.7229, Y 74.9471, Z -3.0000, A 0.000, B 0.000, C 0.000 }
gfCNCPoint2[16429] = {X 140.7395, Y 77.6941, Z -3.0000, A 0.000, B 0.000, C 0.000 }
gfCNCPoint2[16430] = {X 155.7329, Y 61.2293, Z -3.0000, A 0.000, B 0.000, C 0.000 }
gfCNCPoint2[16431] = {X 155.3669, Y 60.5229, Z -3.0000, A 0.000, B 0.000, C 0.000 }
gfCNCPoint2[16432] = {X 155.1393, Y 59.7605, Z -3.0000, A 0.000, B 0.000, C 0.000 }
gfCNCPoint2[16433] = {X 155.0581, Y 58.9691, Z -3.0000, A 0.000, B 0.000, C 0.000 }
gfCNCPoint2[16434] = {X 155.0580, Y 58.0000, Z -3.0000, A 0.000, B 0.000, C 0.000 }
gfCNCPoint2[16435] = {X 155.1643, Y 57.0565, Z -3.0000, A 0.000, B 0.000, C 0.000 }
gfCNCPoint2[16436] = {X 155.4778, Y 56.1603, Z -3.0000, A 0.000, B 0.000, C 0.000 }
gfCNCPoint2[16437] = {X 155.9830, Y 55.3564, Z -3.0000, A 0.000, B 0.000, C 0.000 }
gfCNCPoint2[16438] = {X 156.6544, Y 54.6850, Z -3.0000, A 0.000, B 0.000, C 0.000 }
gfCNCPoint2[16439] = {X 157.4583, Y 54.1799, Z -3.0000, A 0.000, B 0.000, C 0.000 }
gfCNCPoint2[16440] = {X 158.3545, Y 53.8663, Z -3.0000, A 0.000, B 0.000, C 0.000 }
gfCNCPoint2[16441] = {X 159.2980, Y 53.7600, Z -3.0000, A 0.000, B 0.000, C 0.000 }
gfCNCPoint2[16442] = {X 178.5335, Y 53.7600, Z -3.0000, A 0.000, B 0.000, C 0.000 }
gfCNCPoint2[16443] = {X 179.4770, Y 53.8663, Z -3.0000, A 0.000, B 0.000, C 0.000 }
gfCNCPoint2[16444] = {X 180.3732, Y 54.1799, Z -3.0000, A 0.000, B 0.000, C 0.000 }
gfCNCPoint2[16445] = {X 181.1771, Y 54.6850, Z -3.0000, A 0.000, B 0.000, C 0.000 }
gfCNCPoint2[16446] = {X 181.8485, Y 55.3564, Z -3.0000, A 0.000, B 0.000, C 0.000 }
gfCNCPoint2[16447] = {X 182.3536, Y 56.1603, Z -3.0000, A 0.000, B 0.000, C 0.000 }
gfCNCPoint2[16448] = {X 182.6672, Y 57.0565, Z -3.0000, A 0.000, B 0.000, C 0.000 }
gfCNCPoint2[16449] = {X 182.7735, Y 58.0000, Z -3.0000, A 0.000, B 0.000, C 0.000 }
gfCNCPoint2[16450] = {X 182.7735, Y 58.9342, Z -3.0000, A 0.000, B 0.000, C 0.000 }
gfCNCPoint2[16451] = {X 182.6984, Y 59.7286, Z -3.0000, A 0.000, B 0.000, C 0.000 }
gfCNCPoint2[16452] = {X 182.4758, Y 60.4948, Z -3.0000, A 0.000, B 0.000, C 0.000 }
gfCNCPoint2[16453] = {X 182.1136, Y 61.2058, Z -3.0000, A 0.000, B 0.000, C 0.000 }
gfCNCPoint2[16454] = {X 209.4190, Y 91.0080, Z -3.0000, A 0.000, B 0.000, C 0.000 }
gfCNCPoint2[16455] = {X 210.0808, Y 91.6795, Z -3.0000, A 0.000, B 0.000, C 0.000 }
gfCNCPoint2[16456] = {X 210.7899, Y 92.3011, Z -3.0000, A 0.000, B 0.000, C 0.000 }
gfCNCPoint2[16457] = {X 211.0806, Y 92.4849, Z -3.0000, A 0.000, B 0.000, C 0.000 }
gfCNCPoint2[16458] = {X 211.4067, Y 92.5946, Z -3.0000, A 0.000, B 0.000, C 0.000 }
gfCNCPoint2[16459] = {X 213.4016, Y 92.9058, Z -3.0000, A 0.000, B 0.000, C 0.000 }
gfCNCPoint2[16460] = {X 214.4546, Y 92.8166, Z -3.0000, A 0.000, B 0.000, C 0.000 }
gfCNCPoint2[16461] = {X 215.5096, Y 92.7562, Z -3.0000, A 0.000, B 0.000, C 0.000 }
gfCNCPoint2[16462] = {X 216.1940, Y 92.6812, Z -3.0000, A 0.000, B 0.000, C 0.000 }
gfCNCPoint2[16463] = {X 216.8531, Y 92.4818, Z -3.0000, A 0.000, B 0.000, C 0.000 }
gfCNCPoint2[16464] = {X 217.4643, Y 92.1650, Z -3.0000, A 0.000, B 0.000, C 0.000 }
gfCNCPoint2[16465] = {X 223.0046, Y 88.5896, Z -3.0000, A 0.000, B 0.000, C 0.000 }
gfCNCPoint2[16466] = {X 246.0041, Y 73.8823, Z -3.0000, A 0.000, B 0.000, C 0.000 }
gfCNCPoint2[16467] = {X 221.6602, Y 64.3288, Z -3.0000, A 0.000, B 0.000, C 0.000 }
gfCNCPoint2[16468] = {X 219.8842, Y 63.7344, Z -3.0000, A 0.000, B 0.000, C 0.000 }
gfCNCPoint2[16469] = {X 218.0518, Y 63.3470, Z -3.0000, A 0.000, B 0.000, C 0.000 }
gfCNCPoint2[16470] = {X 216.1871, Y 63.1716, Z -3.0000, A 0.000, B 0.000, C 0.000 }
gfCNCPoint2[16471] = {X 215.2725, Y 63.0399, Z -3.0000, A 0.000, B 0.000, C 0.000 }
gfCNCPoint2[16472] = {X 214.4081, Y 62.7131, Z -3.0000, A 0.000, B 0.000, C 0.000 }
gfCNCPoint2[16473] = {X 213.6351, Y 62.2068, Z -3.0000, A 0.000, B 0.000, C 0.000 }
gfCNCPoint2[16474] = {X 212.9901, Y 61.5450, Z -3.0000, A 0.000, B 0.000, C 0.000 }
gfCNCPoint2[16475] = {X 212.5038, Y 60.7593, Z -3.0000, A 0.000, B 0.000, C 0.000 }
gfCNCPoint2[16476] = {X 212.1992, Y 59.8868, Z -3.0000, A 0.000, B 0.000, C 0.000 }
gfCNCPoint2[16477] = {X 212.0910, Y 58.9691, Z -3.0000, A 0.000, B 0.000, C 0.000 }
gfCNCPoint2[16478] = {X 212.0908, Y 58.0000, Z -3.0000, A 0.000, B 0.000, C 0.000 }
gfCNCPoint2[16479] = {X 212.1971, Y 57.0565, Z -3.0000, A 0.000, B 0.000, C 0.000 }
gfCNCPoint2[16480] = {X 212.5107, Y 56.1603, Z -3.0000, A 0.000, B 0.000, C 0.000 }
gfCNCPoint2[16481] = {X 213.0158, Y 55.3564, Z -3.0000, A 0.000, B 0.000, C 0.000 }
gfCNCPoint2[16482] = {X 213.6872, Y 54.6850, Z -3.0000, A 0.000, B 0.000, C 0.000 }
gfCNCPoint2[16483] = {X 214.4911, Y 54.1799, Z -3.0000, A 0.000, B 0.000, C 0.000 }
gfCNCPoint2[16484] = {X 215.3873, Y 53.8663, Z -3.0000, A 0.000, B 0.000, C 0.000 }
gfCNCPoint2[16485] = {X 216.3308, Y 53.7600, Z -3.0000, A 0.000, B 0.000, C 0.000 }
gfCNCPoint2[16486] = {X 237.2617, Y 53.7600, Z -3.0000, A 0.000, B 0.000, C 0.000 }
gfCNCPoint2[16487] = {X 238.2052, Y 53.8663, Z -3.0000, A 0.000, B 0.000, C 0.000 }
gfCNCPoint2[16488] = {X 239.1014, Y 54.1799, Z -3.0000, A 0.000, B 0.000, C 0.000 }
gfCNCPoint2[16489] = {X 239.9053, Y 54.6850, Z -3.0000, A 0.000, B 0.000, C 0.000 }
gfCNCPoint2[16490] = {X 240.5767, Y 55.3564, Z -3.0000, A 0.000, B 0.000, C 0.000 }
gfCNCPoint2[16491] = {X 241.0818, Y 56.1603, Z -3.0000, A 0.000, B 0.000, C 0.000 }
gfCNCPoint2[16492] = {X 241.3954, Y 57.0565, Z -3.0000, A 0.000, B 0.000, C 0.000 }
gfCNCPoint2[16493] = {X 241.5017, Y 58.0000, Z -3.0000, A 0.000, B 0.000, C 0.000 }
gfCNCPoint2[16494] = {X 241.5017, Y 58.2873, Z -3.0000, A 0.000, B 0.000, C 0.000 }
gfCNCPoint2[16495] = {X 247.4591, Y 60.6097, Z -3.0000, A 0.000, B 0.000, C 0.000 }
gfCNCPoint2[16496] = {X 275.7135, Y 71.8205, Z -3.0000, A 0.000, B 0.000, C 0.000 }
gfCNCPoint2[16497] = {X 275.7143, Y 63.1423, Z -3.0000, A 0.000, B 0.000, C 0.000 }
gfCNCPoint2[16498] = {X 274.8656, Y 62.9476, Z -3.0000, A 0.000, B 0.000, C 0.000 }
gfCNCPoint2[16499] = {X 274.0746, Y 62.5838, Z -3.0000, A 0.000, B 0.000, C 0.000 }
gfCNCPoint2[16500] = {X 273.3747, Y 62.0660, Z -3.0000, A 0.000, B 0.000, C 0.000 }
gfCNCPoint2[16501] = {X 272.7952, Y 61.4162, Z -3.0000, A 0.000, B 0.000, C 0.000 }
gfCNCPoint2[16502] = {X 272.3606, Y 60.6617, Z -3.0000, A 0.000, B 0.000, C 0.000 }
gfCNCPoint2[16503] = {X 272.0894, Y 59.8344, Z -3.0000, A 0.000, B 0.000, C 0.000 }
gfCNCPoint2[16504] = {X 271.9928, Y 58.9691, Z -3.0000, A 0.000, B 0.000, C 0.000 }
gfCNCPoint2[16505] = {X 271.9927, Y 58.0000, Z -3.0000, A 0.000, B 0.000, C 0.000 }
gfCNCPoint2[16506] = {X 272.0990, Y 57.0565, Z -3.0000, A 0.000, B 0.000, C 0.000 }
gfCNCPoint2[16507] = {X 272.4126, Y 56.1603, Z -3.0000, A 0.000, B 0.000, C 0.000 }
gfCNCPoint2[16508] = {X 272.9177, Y 55.3564, Z -3.0000, A 0.000, B 0.000, C 0.000 }
gfCNCPoint2[16509] = {X 273.5891, Y 54.6850, Z -3.0000, A 0.000, B 0.000, C 0.000 }
gfCNCPoint2[16510] = {X 274.3930, Y 54.1799, Z -3.0000, A 0.000, B 0.000, C 0.000 }
gfCNCPoint2[16511] = {X 275.2892, Y 53.8663, Z -3.0000, A 0.000, B 0.000, C 0.000 }
gfCNCPoint2[16512] = {X 276.2327, Y 53.7600, Z -3.0000, A 0.000, B 0.000, C 0.000 }
gfCNCPoint2[16513] = {X 292.7731, Y 53.7600, Z -3.0000, A 0.000, B 0.000, C 0.000 }
gfCNCPoint2[16514] = {X 293.7166, Y 53.8663, Z -3.0000, A 0.000, B 0.000, C 0.000 }
gfCNCPoint2[16515] = {X 294.6128, Y 54.1799, Z -3.0000, A 0.000, B 0.000, C 0.000 }
gfCNCPoint2[16516] = {X 295.4167, Y 54.6850, Z -3.0000, A 0.000, B 0.000, C 0.000 }
gfCNCPoint2[16517] = {X 296.0881, Y 55.3564, Z -3.0000, A 0.000, B 0.000, C 0.000 }
gfCNCPoint2[16518] = {X 296.5932, Y 56.1603, Z -3.0000, A 0.000, B 0.000, C 0.000 }
gfCNCPoint2[16519] = {X 296.9068, Y 57.0565, Z -3.0000, A 0.000, B 0.000, C 0.000 }
gfCNCPoint2[16520] = {X 297.0131, Y 58.0000, Z -3.0000, A 0.000, B 0.000, C 0.000 }
gfCNCPoint2[16521] = {X 297.0131, Y 58.9349, Z -3.0000, A 0.000, B 0.000, C 0.000 }
gfCNCPoint2[16522] = {X 296.9203, Y 59.8045, Z -3.0000, A 0.000, B 0.000, C 0.000 }
gfCNCPoint2[16523] = {X 296.6518, Y 60.6369, Z -3.0000, A 0.000, B 0.000, C 0.000 }
gfCNCPoint2[16524] = {X 296.2189, Y 61.3967, Z -3.0000, A 0.000, B 0.000, C 0.000 }
gfCNCPoint2[16525] = {X 295.6398, Y 62.0521, Z -3.0000, A 0.000, B 0.000, C 0.000 }
gfCNCPoint2[16526] = {X 294.9389, Y 62.5753, Z -3.0000, A 0.000, B 0.000, C 0.000 }
gfCNCPoint2[16527] = {X 294.1460, Y 62.9442, Z -3.0000, A 0.000, B 0.000, C 0.000 }
gfCNCPoint2[16528] = {X 293.2944, Y 63.1433, Z -3.0000, A 0.000, B 0.000, C 0.000 }
gfCNCPoint2[16529] = {X 293.3043, Y 92.8512, Z -3.0000, A 0.000, B 0.000, C 0.000 }
gfCNCPoint2[16530] = {X 294.1537, Y 93.0544, Z -3.0000, A 0.000, B 0.000, C 0.000 }
gfCNCPoint2[16531] = {X 294.9440, Y 93.4260, Z -3.0000, A 0.000, B 0.000, C 0.000 }
gfCNCPoint2[16532] = {X 295.6423, Y 93.9506, Z -3.0000, A 0.000, B 0.000, C 0.000 }
gfCNCPoint2[16533] = {X 296.2194, Y 94.6062, Z -3.0000, A 0.000, B 0.000, C 0.000 }
gfCNCPoint2[16534] = {X 296.6511, Y 95.3654, Z -3.0000, A 0.000, B 0.000, C 0.000 }
gfCNCPoint2[16535] = {X 296.9194, Y 96.1965, Z -3.0000, A 0.000, B 0.000, C 0.000 }
gfCNCPoint2[16536] = {X 297.0131, Y 97.0649, Z -3.0000, A 0.000, B 0.000, C 0.000 }
gfCNCPoint2[16537] = {X 297.0131, Y 98.0000, Z -3.0000, A 0.000, B 0.000, C 0.000 }
gfCNCPoint2[16538] = {X 296.9068, Y 98.9435, Z -3.0000, A 0.000, B 0.000, C 0.000 }
gfCNCPoint2[16539] = {X 296.5932, Y 99.8397, Z -3.0000, A 0.000, B 0.000, C 0.000 }
gfCNCPoint2[16540] = {X 296.0881, Y 100.6436, Z -3.0000, A 0.000, B 0.000, C 0.000 }
gfCNCPoint2[16541] = {X 295.4167, Y 101.3150, Z -3.0000, A 0.000, B 0.000, C 0.000 }
gfCNCPoint2[16542] = {X 294.6128, Y 101.8201, Z -3.0000, A 0.000, B 0.000, C 0.000 }
gfCNCPoint2[16543] = {X 293.7166, Y 102.1337, Z -3.0000, A 0.000, B 0.000, C 0.000 }
gfCNCPoint2[16544] = {X 292.7731, Y 102.2400, Z -3.0000, A 0.000, B 0.000, C 0.000 }
gfCNCPoint2[16545] = {X 276.2327, Y 102.2400, Z -3.0000, A 0.000, B 0.000, C 0.000 }
gfCNCPoint2[16546] = {X 275.2892, Y 102.1337, Z -3.0000, A 0.000, B 0.000, C 0.000 }
gfCNCPoint2[16547] = {X 274.3930, Y 101.8201, Z -3.0000, A 0.000, B 0.000, C 0.000 }
gfCNCPoint2[16548] = {X 273.5891, Y 101.3150, Z -3.0000, A 0.000, B 0.000, C 0.000 }
gfCNCPoint2[16549] = {X 272.9177, Y 100.6436, Z -3.0000, A 0.000, B 0.000, C 0.000 }
gfCNCPoint2[16550] = {X 272.4126, Y 99.8397, Z -3.0000, A 0.000, B 0.000, C 0.000 }
gfCNCPoint2[16551] = {X 272.0990, Y 98.9435, Z -3.0000, A 0.000, B 0.000, C 0.000 }
gfCNCPoint2[16552] = {X 271.9927, Y 98.0000, Z -3.0000, A 0.000, B 0.000, C 0.000 }
gfCNCPoint2[16553] = {X 271.9927, Y 97.0659, Z -3.0000, A 0.000, B 0.000, C 0.000 }
gfCNCPoint2[16554] = {X 272.0830, Y 96.1956, Z -3.0000, A 0.000, B 0.000, C 0.000 }
gfCNCPoint2[16555] = {X 272.3500, Y 95.3624, Z -3.0000, A 0.000, B 0.000, C 0.000 }
gfCNCPoint2[16556] = {X 272.7823, Y 94.6018, Z -3.0000, A 0.000, B 0.000, C 0.000 }
gfCNCPoint2[16557] = {X 273.3615, Y 93.9460, Z -3.0000, A 0.000, B 0.000, C 0.000 }
gfCNCPoint2[16558] = {X 274.0630, Y 93.4231, Z -3.0000, A 0.000, B 0.000, C 0.000 }
gfCNCPoint2[16559] = {X 274.8569, Y 93.0553, Z -3.0000, A 0.000, B 0.000, C 0.000 }
gfCNCPoint2[16560] = {X 275.7094, Y 92.8584, Z -3.0000, A 0.000, B 0.000, C 0.000 }
gfCNCPoint2[16561] = {X 275.7094, Y 85.5404, Z -3.0000, A 0.000, B 0.000, C 0.000 }
gfCNCPoint2[16562] = {X 262.6311, Y 80.4137, Z -3.0000, A 0.000, B 0.000, C 0.000 }
gfCNCPoint2[16563] = {X 262.2333, Y 80.6642, Z -3.0000, A 0.000, B 0.000, C 0.000 }
gfCNCPoint2[16564] = {X 237.7158, Y 96.5447, Z -3.0000, A 0.000, B 0.000, C 0.000 }
gfCNCPoint2[16565] = {X 237.7198, Y 97.0650, Z -3.0000, A 0.000, B 0.000, C 0.000 }
gfCNCPoint2[16566] = {X 237.7198, Y 98.0000, Z -3.0000, A 0.000, B 0.000, C 0.000 }
gfCNCPoint2[16567] = {X 237.6135, Y 98.9435, Z -3.0000, A 0.000, B 0.000, C 0.000 }
gfCNCPoint2[16568] = {X 237.2999, Y 99.8397, Z -3.0000, A 0.000, B 0.000, C 0.000 }
gfCNCPoint2[16569] = {X 236.7948, Y 100.6436, Z -3.0000, A 0.000, B 0.000, C 0.000 }
gfCNCPoint2[16570] = {X 236.1234, Y 101.3150, Z -3.0000, A 0.000, B 0.000, C 0.000 }
gfCNCPoint2[16571] = {X 235.3195, Y 101.8201, Z -3.0000, A 0.000, B 0.000, C 0.000 }
gfCNCPoint2[16572] = {X 234.4233, Y 102.1337, Z -3.0000, A 0.000, B 0.000, C 0.000 }
gfCNCPoint2[16573] = {X 233.4798, Y 102.2400, Z -3.0000, A 0.000, B 0.000, C 0.000 }
gfCNCPoint2[16574] = {X 214.1790, Y 102.2400, Z -3.0000, A 0.000, B 0.000, C 0.000 }
gfCNCPoint2[16575] = {X 213.7861, Y 102.2218, Z -3.0000, A 0.000, B 0.000, C 0.000 }
gfCNCPoint2[16576] = {X 213.3966, Y 102.1672, Z -3.0000, A 0.000, B 0.000, C 0.000 }
gfCNCPoint2[16577] = {X 213.0070, Y 102.2218, Z -3.0000, A 0.000, B 0.000, C 0.000 }
gfCNCPoint2[16578] = {X 212.6141, Y 102.2400, Z -3.0000, A 0.000, B 0.000, C 0.000 }
gfCNCPoint2[16579] = {X 194.9870, Y 102.2400, Z -3.0000, A 0.000, B 0.000, C 0.000 }
gfCNCPoint2[16580] = {X 194.0435, Y 102.1337, Z -3.0000, A 0.000, B 0.000, C 0.000 }
gfCNCPoint2[16581] = {X 193.1473, Y 101.8201, Z -3.0000, A 0.000, B 0.000, C 0.000 }
gfCNCPoint2[16582] = {X 192.3434, Y 101.3150, Z -3.0000, A 0.000, B 0.000, C 0.000 }
gfCNCPoint2[16583] = {X 191.6720, Y 100.6436, Z -3.0000, A 0.000, B 0.000, C 0.000 }
gfCNCPoint2[16584] = {X 191.1669, Y 99.8397, Z -3.0000, A 0.000, B 0.000, C 0.000 }
gfCNCPoint2[16585] = {X 190.8533, Y 98.9435, Z -3.0000, A 0.000, B 0.000, C 0.000 }
gfCNCPoint2[16586] = {X 190.7470, Y 98.0000, Z -3.0000, A 0.000, B 0.000, C 0.000 }
gfCNCPoint2[16587] = {X 190.7470, Y 97.0659, Z -3.0000, A 0.000, B 0.000, C 0.000 }
gfCNCPoint2[16588] = {X 190.8557, Y 96.1118, Z -3.0000, A 0.000, B 0.000, C 0.000 }
gfCNCPoint2[16589] = {X 191.1764, Y 95.2065, Z -3.0000, A 0.000, B 0.000, C 0.000 }
gfCNCPoint2[16590] = {X 191.6926, Y 94.3967, Z -3.0000, A 0.000, B 0.000, C 0.000 }
gfCNCPoint2[16591] = {X 188.5999, Y 91.0202, Z -3.0000, A 0.000, B 0.000, C 0.000 }
gfCNCPoint2[16592] = {X 150.0543, Y 91.0202, Z -3.0000, A 0.000, B 0.000, C 0.000 }
gfCNCPoint2[16593] = {X 147.0393, Y 94.3604, Z -3.0000, A 0.000, B 0.000, C 0.000 }
gfCNCPoint2[16594] = {X 147.5714, Y 95.1785, Z -3.0000, A 0.000, B 0.000, C 0.000 }
gfCNCPoint2[16595] = {X 147.9038, Y 96.0961, Z -3.0000, A 0.000, B 0.000, C 0.000 }
gfCNCPoint2[16596] = {X 148.0191, Y 97.0652, Z -3.0000, A 0.000, B 0.000, C 0.000 }
gfCNCPoint2[16597] = {X 148.0191, Y 98.0000, Z -3.0000, A 0.000, B 0.000, C 0.000 }
gfCNCPoint2[16598] = {X 147.9128, Y 98.9435, Z -3.0000, A 0.000, B 0.000, C 0.000 }
gfCNCPoint2[16599] = {X 147.5992, Y 99.8397, Z -3.0000, A 0.000, B 0.000, C 0.000 }
gfCNCPoint2[16600] = {X 147.0941, Y 100.6436, Z -3.0000, A 0.000, B 0.000, C 0.000 }
gfCNCPoint2[16601] = {X 146.4227, Y 101.3150, Z -3.0000, A 0.000, B 0.000, C 0.000 }
gfCNCPoint2[16602] = {X 145.6188, Y 101.8201, Z -3.0000, A 0.000, B 0.000, C 0.000 }
gfCNCPoint2[16603] = {X 144.7226, Y 102.1337, Z -3.0000, A 0.000, B 0.000, C 0.000 }
gfCNCPoint2[16604] = {X 143.7791, Y 102.2400, Z -3.0000, A 0.000, B 0.000, C 0.000 }
gfCNCPoint2[16605] = {X 125.0000, Y 102.2400, Z -3.0000, A 0.000, B 0.000, C 0.000 }
gfCNCPoint2[16606] = {X 124.0565, Y 102.1337, Z -3.0000, A 0.000, B 0.000, C 0.000 }
gfCNCPoint2[16607] = {X 123.1603, Y 101.8201, Z -3.0000, A 0.000, B 0.000, C 0.000 }
gfCNCPoint2[16608] = {X 122.3564, Y 101.3150, Z -3.0000, A 0.000, B 0.000, C 0.000 }
gfCNCPoint2[16609] = {X 121.6850, Y 100.6436, Z -3.0000, A 0.000, B 0.000, C 0.000 }
gfCNCPoint2[16610] = {X 121.1799, Y 99.8397, Z -3.0000, A 0.000, B 0.000, C 0.000 }
gfCNCPoint2[16611] = {X 120.8663, Y 98.9435, Z -3.0000, A 0.000, B 0.000, C 0.000 }
gfCNCPoint2[16612] = {X 120.7600, Y 98.0000, Z -3.0000, A 0.000, B 0.000, C 0.000 }
gfCNCPoint2[16613] = {X 120.7600, Y 97.0659, Z -3.0000, A 0.000, B 0.000, C 0.000 }
gfCNCPoint2[16614] = {X 120.8619, Y 96.1421, Z -3.0000, A 0.000, B 0.000, C 0.000 }
gfCNCPoint2[16615] = {X 121.1626, Y 95.2626, Z -3.0000, A 0.000, B 0.000, C 0.000 }
gfCNCPoint2[16616] = {X 121.6478, Y 94.4698, Z -3.0000, A 0.000, B 0.000, C 0.000 }
gfCNCPoint2[16617] = {X 122.2940, Y 93.8017, Z -3.0000, A 0.000, B 0.000, C 0.000 }
gfCNCPoint2[16618] = {X 123.0703, Y 93.2905, Z -3.0000, A 0.000, B 0.000, C 0.000 }
gfCNCPoint2[16619] = {X 123.9393, Y 92.9608, Z -3.0000, A 0.000, B 0.000, C 0.000 }
gfCNCPoint2[16620] = {X 124.8593, Y 92.8283, Z -3.0000, A 0.000, B 0.000, C 0.000 }
gfCNCPoint2[16621] = {X 124.8983, Y 92.8112, Z -3.0000, A 0.000, B 0.000, C 0.000 }
gfCNCPoint2[16622] = {X 124.9397, Y 92.8013, Z -3.0000, A 0.000, B 0.000, C 0.000 }
gfCNCPoint2[16623] = {X 125.4604, Y 92.7240, Z -3.0000, A 0.000, B 0.000, C 0.000 }
gfCNCPoint2[16624] = {X 126.3060, Y 92.5808, Z -3.0000, A 0.000, B 0.000, C 0.000 }
gfCNCPoint2[16625] = {X 127.1399, Y 92.3804, Z -3.0000, A 0.000, B 0.000, C 0.000 }
gfCNCPoint2[16626] = {X 128.3720, Y 91.2198, Z -3.0000, A 0.000, B 0.000, C 0.000 }
gfCNCPoint2[16627] = {X 129.5390, Y 89.9938, Z -3.0000, A 0.000, B 0.000, C 0.000 }
gfCNCPoint2[16628] = {X 140.7395, Y 77.6941, Z -3.0000, A 0.000, B 0.000, C 0.000 }
gfCNCPoint2[16629] = {X 137.7820, Y 75.0009, Z -3.0000, A 0.000, B 0.000, C 0.000 }
gfCNCPoint2[16630] = {X 140.7987, Y 77.7480, Z -3.0000, A 0.000, B 0.000, C 0.000 }
gfCNCPoint2[16631] = {X 155.8338, Y 61.2374, Z -3.0000, A 0.000, B 0.000, C 0.000 }
gfCNCPoint2[16632] = {X 155.4566, Y 60.5308, Z -3.0000, A 0.000, B 0.000, C 0.000 }
gfCNCPoint2[16633] = {X 155.2218, Y 59.7650, Z -3.0000, A 0.000, B 0.000, C 0.000 }
gfCNCPoint2[16634] = {X 155.1381, Y 58.9684, Z -3.0000, A 0.000, B 0.000, C 0.000 }
gfCNCPoint2[16635] = {X 155.1380, Y 58.0000, Z -3.0000, A 0.000, B 0.000, C 0.000 }
gfCNCPoint2[16636] = {X 155.2423, Y 57.0743, Z -3.0000, A 0.000, B 0.000, C 0.000 }
gfCNCPoint2[16637] = {X 155.5499, Y 56.1950, Z -3.0000, A 0.000, B 0.000, C 0.000 }
gfCNCPoint2[16638] = {X 156.0455, Y 55.4063, Z -3.0000, A 0.000, B 0.000, C 0.000 }
gfCNCPoint2[16639] = {X 156.7042, Y 54.7476, Z -3.0000, A 0.000, B 0.000, C 0.000 }
gfCNCPoint2[16640] = {X 157.4930, Y 54.2520, Z -3.0000, A 0.000, B 0.000, C 0.000 }
gfCNCPoint2[16641] = {X 158.3723, Y 53.9443, Z -3.0000, A 0.000, B 0.000, C 0.000 }
gfCNCPoint2[16642] = {X 159.2980, Y 53.8400, Z -3.0000, A 0.000, B 0.000, C 0.000 }
gfCNCPoint2[16643] = {X 178.5335, Y 53.8400, Z -3.0000, A 0.000, B 0.000, C 0.000 }
gfCNCPoint2[16644] = {X 179.4592, Y 53.9443, Z -3.0000, A 0.000, B 0.000, C 0.000 }
gfCNCPoint2[16645] = {X 180.3385, Y 54.2520, Z -3.0000, A 0.000, B 0.000, C 0.000 }
gfCNCPoint2[16646] = {X 181.1272, Y 54.7476, Z -3.0000, A 0.000, B 0.000, C 0.000 }
gfCNCPoint2[16647] = {X 181.7859, Y 55.4063, Z -3.0000, A 0.000, B 0.000, C 0.000 }
gfCNCPoint2[16648] = {X 182.2815, Y 56.1950, Z -3.0000, A 0.000, B 0.000, C 0.000 }
gfCNCPoint2[16649] = {X 182.5892, Y 57.0743, Z -3.0000, A 0.000, B 0.000, C 0.000 }
gfCNCPoint2[16650] = {X 182.6935, Y 58.0000, Z -3.0000, A 0.000, B 0.000, C 0.000 }
gfCNCPoint2[16651] = {X 182.6935, Y 58.9342, Z -3.0000, A 0.000, B 0.000, C 0.000 }
gfCNCPoint2[16652] = {X 182.6159, Y 59.7336, Z -3.0000, A 0.000, B 0.000, C 0.000 }
gfCNCPoint2[16653] = {X 182.3862, Y 60.5032, Z -3.0000, A 0.000, B 0.000, C 0.000 }
gfCNCPoint2[16654] = {X 182.0129, Y 61.2143, Z -3.0000, A 0.000, B 0.000, C 0.000 }
gfCNCPoint2[16655] = {X 209.3600, Y 91.0621, Z -3.0000, A 0.000, B 0.000, C 0.000 }
gfCNCPoint2[16656] = {X 210.0260, Y 91.7377, Z -3.0000, A 0.000, B 0.000, C 0.000 }
gfCNCPoint2[16657] = {X 210.7394, Y 92.3631, Z -3.0000, A 0.000, B 0.000, C 0.000 }
gfCNCPoint2[16658] = {X 211.0472, Y 92.5576, Z -3.0000, A 0.000, B 0.000, C 0.000 }
gfCNCPoint2[16659] = {X 211.3924, Y 92.6734, Z -3.0000, A 0.000, B 0.000, C 0.000 }
gfCNCPoint2[16660] = {X 213.3993, Y 92.9864, Z -3.0000, A 0.000, B 0.000, C 0.000 }
gfCNCPoint2[16661] = {X 214.4547, Y 92.8968, Z -3.0000, A 0.000, B 0.000, C 0.000 }
gfCNCPoint2[16662] = {X 215.5121, Y 92.8362, Z -3.0000, A 0.000, B 0.000, C 0.000 }
gfCNCPoint2[16663] = {X 216.2108, Y 92.7594, Z -3.0000, A 0.000, B 0.000, C 0.000 }
gfCNCPoint2[16664] = {X 216.8836, Y 92.5558, Z -3.0000, A 0.000, B 0.000, C 0.000 }
gfCNCPoint2[16665] = {X 217.5077, Y 92.2322, Z -3.0000, A 0.000, B 0.000, C 0.000 }
gfCNCPoint2[16666] = {X 223.0478, Y 88.6569, Z -3.0000, A 0.000, B 0.000, C 0.000 }
gfCNCPoint2[16667] = {X 246.1794, Y 73.8652, Z -3.0000, A 0.000, B 0.000, C 0.000 }
gfCNCPoint2[16668] = {X 221.6899, Y 64.2545, Z -3.0000, A 0.000, B 0.000, C 0.000 }
gfCNCPoint2[16669] = {X 219.9052, Y 63.6572, Z -3.0000, A 0.000, B 0.000, C 0.000 }
gfCNCPoint2[16670] = {X 218.0638, Y 63.2679, Z -3.0000, A 0.000, B 0.000, C 0.000 }
gfCNCPoint2[16671] = {X 216.1900, Y 63.0917, Z -3.0000, A 0.000, B 0.000, C 0.000 }
gfCNCPoint2[16672] = {X 215.2926, Y 62.9624, Z -3.0000, A 0.000, B 0.000, C 0.000 }
gfCNCPoint2[16673] = {X 214.4445, Y 62.6418, Z -3.0000, A 0.000, B 0.000, C 0.000 }
gfCNCPoint2[16674] = {X 213.6860, Y 62.1451, Z -3.0000, A 0.000, B 0.000, C 0.000 }
gfCNCPoint2[16675] = {X 213.0532, Y 61.4958, Z -3.0000, A 0.000, B 0.000, C 0.000 }
gfCNCPoint2[16676] = {X 212.5760, Y 60.7249, Z -3.0000, A 0.000, B 0.000, C 0.000 }
gfCNCPoint2[16677] = {X 212.2772, Y 59.8688, Z -3.0000, A 0.000, B 0.000, C 0.000 }
gfCNCPoint2[16678] = {X 212.1710, Y 58.9684, Z -3.0000, A 0.000, B 0.000, C 0.000 }
gfCNCPoint2[16679] = {X 212.1708, Y 58.0000, Z -3.0000, A 0.000, B 0.000, C 0.000 }
gfCNCPoint2[16680] = {X 212.2751, Y 57.0743, Z -3.0000, A 0.000, B 0.000, C 0.000 }
gfCNCPoint2[16681] = {X 212.5828, Y 56.1950, Z -3.0000, A 0.000, B 0.000, C 0.000 }
gfCNCPoint2[16682] = {X 213.0784, Y 55.4063, Z -3.0000, A 0.000, B 0.000, C 0.000 }
gfCNCPoint2[16683] = {X 213.7371, Y 54.7476, Z -3.0000, A 0.000, B 0.000, C 0.000 }
gfCNCPoint2[16684] = {X 214.5259, Y 54.2520, Z -3.0000, A 0.000, B 0.000, C 0.000 }
gfCNCPoint2[16685] = {X 215.4051, Y 53.9443, Z -3.0000, A 0.000, B 0.000, C 0.000 }
gfCNCPoint2[16686] = {X 216.3308, Y 53.8400, Z -3.0000, A 0.000, B 0.000, C 0.000 }
gfCNCPoint2[16687] = {X 237.2617, Y 53.8400, Z -3.0000, A 0.000, B 0.000, C 0.000 }
gfCNCPoint2[16688] = {X 238.1874, Y 53.9443, Z -3.0000, A 0.000, B 0.000, C 0.000 }
gfCNCPoint2[16689] = {X 239.0666, Y 54.2520, Z -3.0000, A 0.000, B 0.000, C 0.000 }
gfCNCPoint2[16690] = {X 239.8554, Y 54.7476, Z -3.0000, A 0.000, B 0.000, C 0.000 }
gfCNCPoint2[16691] = {X 240.5141, Y 55.4063, Z -3.0000, A 0.000, B 0.000, C 0.000 }
gfCNCPoint2[16692] = {X 241.0097, Y 56.1950, Z -3.0000, A 0.000, B 0.000, C 0.000 }
gfCNCPoint2[16693] = {X 241.3174, Y 57.0743, Z -3.0000, A 0.000, B 0.000, C 0.000 }
gfCNCPoint2[16694] = {X 241.4217, Y 58.0000, Z -3.0000, A 0.000, B 0.000, C 0.000 }
gfCNCPoint2[16695] = {X 241.4217, Y 58.3420, Z -3.0000, A 0.000, B 0.000, C 0.000 }
gfCNCPoint2[16696] = {X 247.4298, Y 60.6842, Z -3.0000, A 0.000, B 0.000, C 0.000 }
gfCNCPoint2[16697] = {X 275.7935, Y 71.9383, Z -3.0000, A 0.000, B 0.000, C 0.000 }
gfCNCPoint2[16698] = {X 275.7943, Y 63.0709, Z -3.0000, A 0.000, B 0.000, C 0.000 }
gfCNCPoint2[16699] = {X 275.6919, Y 63.0588, Z -3.0000, A 0.000, B 0.000, C 0.000 }
gfCNCPoint2[16700] = {X 275.5899, Y 63.0441, Z -3.0000, A 0.000, B 0.000, C 0.000 }
gfCNCPoint2[16701] = {X 274.6522, Y 62.7821, Z -3.0000, A 0.000, B 0.000, C 0.000 }
gfCNCPoint2[16702] = {X 273.8011, Y 62.3094, Z -3.0000, A 0.000, B 0.000, C 0.000 }
gfCNCPoint2[16703] = {X 273.0832, Y 61.6519, Z -3.0000, A 0.000, B 0.000, C 0.000 }
gfCNCPoint2[16704] = {X 272.5378, Y 60.8454, Z -3.0000, A 0.000, B 0.000, C 0.000 }
gfCNCPoint2[16705] = {X 272.1947, Y 59.9343, Z -3.0000, A 0.000, B 0.000, C 0.000 }
gfCNCPoint2[16706] = {X 272.0728, Y 58.9684, Z -3.0000, A 0.000, B 0.000, C 0.000 }
gfCNCPoint2[16707] = {X 272.0727, Y 58.0000, Z -3.0000, A 0.000, B 0.000, C 0.000 }
gfCNCPoint2[16708] = {X 272.1770, Y 57.0743, Z -3.0000, A 0.000, B 0.000, C 0.000 }
gfCNCPoint2[16709] = {X 272.4847, Y 56.1950, Z -3.0000, A 0.000, B 0.000, C 0.000 }
gfCNCPoint2[16710] = {X 272.9803, Y 55.4063, Z -3.0000, A 0.000, B 0.000, C 0.000 }
gfCNCPoint2[16711] = {X 273.6390, Y 54.7476, Z -3.0000, A 0.000, B 0.000, C 0.000 }
gfCNCPoint2[16712] = {X 274.4277, Y 54.2520, Z -3.0000, A 0.000, B 0.000, C 0.000 }
gfCNCPoint2[16713] = {X 275.3070, Y 53.9443, Z -3.0000, A 0.000, B 0.000, C 0.000 }
gfCNCPoint2[16714] = {X 276.2327, Y 53.8400, Z -3.0000, A 0.000, B 0.000, C 0.000 }
gfCNCPoint2[16715] = {X 292.7731, Y 53.8400, Z -3.0000, A 0.000, B 0.000, C 0.000 }
gfCNCPoint2[16716] = {X 293.6988, Y 53.9443, Z -3.0000, A 0.000, B 0.000, C 0.000 }
gfCNCPoint2[16717] = {X 294.5780, Y 54.2520, Z -3.0000, A 0.000, B 0.000, C 0.000 }
gfCNCPoint2[16718] = {X 295.3668, Y 54.7476, Z -3.0000, A 0.000, B 0.000, C 0.000 }
gfCNCPoint2[16719] = {X 296.0255, Y 55.4063, Z -3.0000, A 0.000, B 0.000, C 0.000 }
gfCNCPoint2[16720] = {X 296.5211, Y 56.1950, Z -3.0000, A 0.000, B 0.000, C 0.000 }
gfCNCPoint2[16721] = {X 296.8288, Y 57.0743, Z -3.0000, A 0.000, B 0.000, C 0.000 }
gfCNCPoint2[16722] = {X 296.9331, Y 58.0000, Z -3.0000, A 0.000, B 0.000, C 0.000 }
gfCNCPoint2[16723] = {X 296.9331, Y 58.9346, Z -3.0000, A 0.000, B 0.000, C 0.000 }
gfCNCPoint2[16724] = {X 296.8152, Y 59.9063, Z -3.0000, A 0.000, B 0.000, C 0.000 }
gfCNCPoint2[16725] = {X 296.4743, Y 60.8238, Z -3.0000, A 0.000, B 0.000, C 0.000 }
gfCNCPoint2[16726] = {X 295.9293, Y 61.6368, Z -3.0000, A 0.000, B 0.000, C 0.000 }
gfCNCPoint2[16727] = {X 295.2101, Y 62.3007, Z -3.0000, A 0.000, B 0.000, C 0.000 }
gfCNCPoint2[16728] = {X 294.3561, Y 62.7789, Z -3.0000, A 0.000, B 0.000, C 0.000 }
gfCNCPoint2[16729] = {X 293.4143, Y 63.0453, Z -3.0000, A 0.000, B 0.000, C 0.000 }
gfCNCPoint2[16730] = {X 293.3179, Y 63.0595, Z -3.0000, A 0.000, B 0.000, C 0.000 }
gfCNCPoint2[16731] = {X 293.2212, Y 63.0715, Z -3.0000, A 0.000, B 0.000, C 0.000 }
gfCNCPoint2[16732] = {X 293.2121, Y 63.1621, Z -3.0000, A 0.000, B 0.000, C 0.000 }
gfCNCPoint2[16733] = {X 293.2243, Y 92.9219, Z -3.0000, A 0.000, B 0.000, C 0.000 }
gfCNCPoint2[16734] = {X 293.3191, Y 92.9340, Z -3.0000, A 0.000, B 0.000, C 0.000 }
gfCNCPoint2[16735] = {X 293.4136, Y 92.9483, Z -3.0000, A 0.000, B 0.000, C 0.000 }
gfCNCPoint2[16736] = {X 294.3550, Y 93.2173, Z -3.0000, A 0.000, B 0.000, C 0.000 }
gfCNCPoint2[16737] = {X 295.2085, Y 93.6973, Z -3.0000, A 0.000, B 0.000, C 0.000 }
gfCNCPoint2[16738] = {X 295.9273, Y 94.3622, Z -3.0000, A 0.000, B 0.000, C 0.000 }
gfCNCPoint2[16739] = {X 296.4723, Y 95.1757, Z -3.0000, A 0.000, B 0.000, C 0.000 }
gfCNCPoint2[16740] = {X 296.8138, Y 96.0934, Z -3.0000, A 0.000, B 0.000, C 0.000 }
gfCNCPoint2[16741] = {X 296.9331, Y 97.0653, Z -3.0000, A 0.000, B 0.000, C 0.000 }
gfCNCPoint2[16742] = {X 296.9331, Y 98.0000, Z -3.0000, A 0.000, B 0.000, C 0.000 }
gfCNCPoint2[16743] = {X 296.8288, Y 98.9257, Z -3.0000, A 0.000, B 0.000, C 0.000 }
gfCNCPoint2[16744] = {X 296.5211, Y 99.8050, Z -3.0000, A 0.000, B 0.000, C 0.000 }
gfCNCPoint2[16745] = {X 296.0255, Y 100.5937, Z -3.0000, A 0.000, B 0.000, C 0.000 }
gfCNCPoint2[16746] = {X 295.3668, Y 101.2524, Z -3.0000, A 0.000, B 0.000, C 0.000 }
gfCNCPoint2[16747] = {X 294.5780, Y 101.7480, Z -3.0000, A 0.000, B 0.000, C 0.000 }
gfCNCPoint2[16748] = {X 293.6988, Y 102.0557, Z -3.0000, A 0.000, B 0.000, C 0.000 }
gfCNCPoint2[16749] = {X 292.7731, Y 102.1600, Z -3.0000, A 0.000, B 0.000, C 0.000 }
gfCNCPoint2[16750] = {X 276.2327, Y 102.1600, Z -3.0000, A 0.000, B 0.000, C 0.000 }
gfCNCPoint2[16751] = {X 275.3070, Y 102.0557, Z -3.0000, A 0.000, B 0.000, C 0.000 }
gfCNCPoint2[16752] = {X 274.4277, Y 101.7480, Z -3.0000, A 0.000, B 0.000, C 0.000 }
gfCNCPoint2[16753] = {X 273.6390, Y 101.2524, Z -3.0000, A 0.000, B 0.000, C 0.000 }
gfCNCPoint2[16754] = {X 272.9803, Y 100.5937, Z -3.0000, A 0.000, B 0.000, C 0.000 }
gfCNCPoint2[16755] = {X 272.4847, Y 99.8050, Z -3.0000, A 0.000, B 0.000, C 0.000 }
gfCNCPoint2[16756] = {X 272.1770, Y 98.9257, Z -3.0000, A 0.000, B 0.000, C 0.000 }
gfCNCPoint2[16757] = {X 272.0727, Y 98.0000, Z -3.0000, A 0.000, B 0.000, C 0.000 }
gfCNCPoint2[16758] = {X 272.0727, Y 97.0659, Z -3.0000, A 0.000, B 0.000, C 0.000 }
gfCNCPoint2[16759] = {X 272.1633, Y 96.2022, Z -3.0000, A 0.000, B 0.000, C 0.000 }
gfCNCPoint2[16760] = {X 272.4314, Y 95.3761, Z -3.0000, A 0.000, B 0.000, C 0.000 }
gfCNCPoint2[16761] = {X 272.8650, Y 94.6237, Z -3.0000, A 0.000, B 0.000, C 0.000 }
gfCNCPoint2[16762] = {X 273.4455, Y 93.9777, Z -3.0000, A 0.000, B 0.000, C 0.000 }
gfCNCPoint2[16763] = {X 274.1474, Y 93.4663, Z -3.0000, A 0.000, B 0.000, C 0.000 }
gfCNCPoint2[16764] = {X 274.9402, Y 93.1118, Z -3.0000, A 0.000, B 0.000, C 0.000 }
gfCNCPoint2[16765] = {X 275.7894, Y 92.9296, Z -3.0000, A 0.000, B 0.000, C 0.000 }
gfCNCPoint2[16766] = {X 275.7894, Y 85.4858, Z -3.0000, A 0.000, B 0.000, C 0.000 }
gfCNCPoint2[16767] = {X 262.6227, Y 80.3245, Z -3.0000, A 0.000, B 0.000, C 0.000 }
gfCNCPoint2[16768] = {X 262.1902, Y 80.5968, Z -3.0000, A 0.000, B 0.000, C 0.000 }
gfCNCPoint2[16769] = {X 237.6355, Y 96.5014, Z -3.0000, A 0.000, B 0.000, C 0.000 }
gfCNCPoint2[16770] = {X 237.6398, Y 97.0653, Z -3.0000, A 0.000, B 0.000, C 0.000 }
gfCNCPoint2[16771] = {X 237.6398, Y 98.0000, Z -3.0000, A 0.000, B 0.000, C 0.000 }
gfCNCPoint2[16772] = {X 237.5355, Y 98.9257, Z -3.0000, A 0.000, B 0.000, C 0.000 }
gfCNCPoint2[16773] = {X 237.2278, Y 99.8050, Z -3.0000, A 0.000, B 0.000, C 0.000 }
gfCNCPoint2[16774] = {X 236.7322, Y 100.5937, Z -3.0000, A 0.000, B 0.000, C 0.000 }
gfCNCPoint2[16775] = {X 236.0735, Y 101.2524, Z -3.0000, A 0.000, B 0.000, C 0.000 }
gfCNCPoint2[16776] = {X 235.2847, Y 101.7480, Z -3.0000, A 0.000, B 0.000, C 0.000 }
gfCNCPoint2[16777] = {X 234.4055, Y 102.0557, Z -3.0000, A 0.000, B 0.000, C 0.000 }
gfCNCPoint2[16778] = {X 233.4798, Y 102.1600, Z -3.0000, A 0.000, B 0.000, C 0.000 }
gfCNCPoint2[16779] = {X 214.1790, Y 102.1600, Z -3.0000, A 0.000, B 0.000, C 0.000 }
gfCNCPoint2[16780] = {X 213.7860, Y 102.1414, Z -3.0000, A 0.000, B 0.000, C 0.000 }
gfCNCPoint2[16781] = {X 213.3966, Y 102.0857, Z -3.0000, A 0.000, B 0.000, C 0.000 }
gfCNCPoint2[16782] = {X 213.0071, Y 102.1414, Z -3.0000, A 0.000, B 0.000, C 0.000 }
gfCNCPoint2[16783] = {X 212.6141, Y 102.1600, Z -3.0000, A 0.000, B 0.000, C 0.000 }
gfCNCPoint2[16784] = {X 194.9870, Y 102.1600, Z -3.0000, A 0.000, B 0.000, C 0.000 }
gfCNCPoint2[16785] = {X 194.0613, Y 102.0557, Z -3.0000, A 0.000, B 0.000, C 0.000 }
gfCNCPoint2[16786] = {X 193.1820, Y 101.7480, Z -3.0000, A 0.000, B 0.000, C 0.000 }
gfCNCPoint2[16787] = {X 192.3932, Y 101.2524, Z -3.0000, A 0.000, B 0.000, C 0.000 }
gfCNCPoint2[16788] = {X 191.7345, Y 100.5937, Z -3.0000, A 0.000, B 0.000, C 0.000 }
gfCNCPoint2[16789] = {X 191.2389, Y 99.8050, Z -3.0000, A 0.000, B 0.000, C 0.000 }
gfCNCPoint2[16790] = {X 190.9313, Y 98.9257, Z -3.0000, A 0.000, B 0.000, C 0.000 }
gfCNCPoint2[16791] = {X 190.8270, Y 98.0000, Z -3.0000, A 0.000, B 0.000, C 0.000 }
gfCNCPoint2[16792] = {X 190.8270, Y 97.0659, Z -3.0000, A 0.000, B 0.000, C 0.000 }
gfCNCPoint2[16793] = {X 190.9241, Y 96.1723, Z -3.0000, A 0.000, B 0.000, C 0.000 }
gfCNCPoint2[16794] = {X 191.2109, Y 95.3203, Z -3.0000, A 0.000, B 0.000, C 0.000 }
gfCNCPoint2[16795] = {X 191.6741, Y 94.5499, Z -3.0000, A 0.000, B 0.000, C 0.000 }
gfCNCPoint2[16796] = {X 191.7354, Y 94.4712, Z -3.0000, A 0.000, B 0.000, C 0.000 }
gfCNCPoint2[16797] = {X 191.7986, Y 94.3939, Z -3.0000, A 0.000, B 0.000, C 0.000 }
gfCNCPoint2[16798] = {X 188.6351, Y 90.9402, Z -3.0000, A 0.000, B 0.000, C 0.000 }
gfCNCPoint2[16799] = {X 150.0187, Y 90.9402, Z -3.0000, A 0.000, B 0.000, C 0.000 }
gfCNCPoint2[16800] = {X 146.9332, Y 94.3586, Z -3.0000, A 0.000, B 0.000, C 0.000 }
gfCNCPoint2[16801] = {X 147.4790, Y 95.1731, Z -3.0000, A 0.000, B 0.000, C 0.000 }
gfCNCPoint2[16802] = {X 147.8206, Y 96.0922, Z -3.0000, A 0.000, B 0.000, C 0.000 }
gfCNCPoint2[16803] = {X 147.9391, Y 97.0655, Z -3.0000, A 0.000, B 0.000, C 0.000 }
gfCNCPoint2[16804] = {X 147.9391, Y 98.0000, Z -3.0000, A 0.000, B 0.000, C 0.000 }
gfCNCPoint2[16805] = {X 147.8348, Y 98.9257, Z -3.0000, A 0.000, B 0.000, C 0.000 }
gfCNCPoint2[16806] = {X 147.5271, Y 99.8050, Z -3.0000, A 0.000, B 0.000, C 0.000 }
gfCNCPoint2[16807] = {X 147.0315, Y 100.5937, Z -3.0000, A 0.000, B 0.000, C 0.000 }
gfCNCPoint2[16808] = {X 146.3728, Y 101.2524, Z -3.0000, A 0.000, B 0.000, C 0.000 }
gfCNCPoint2[16809] = {X 145.5841, Y 101.7480, Z -3.0000, A 0.000, B 0.000, C 0.000 }
gfCNCPoint2[16810] = {X 144.7048, Y 102.0557, Z -3.0000, A 0.000, B 0.000, C 0.000 }
gfCNCPoint2[16811] = {X 143.7791, Y 102.1600, Z -3.0000, A 0.000, B 0.000, C 0.000 }
gfCNCPoint2[16812] = {X 125.0000, Y 102.1600, Z -3.0000, A 0.000, B 0.000, C 0.000 }
gfCNCPoint2[16813] = {X 124.0743, Y 102.0557, Z -3.0000, A 0.000, B 0.000, C 0.000 }
gfCNCPoint2[16814] = {X 123.1950, Y 101.7480, Z -3.0000, A 0.000, B 0.000, C 0.000 }
gfCNCPoint2[16815] = {X 122.4063, Y 101.2524, Z -3.0000, A 0.000, B 0.000, C 0.000 }
gfCNCPoint2[16816] = {X 121.7476, Y 100.5937, Z -3.0000, A 0.000, B 0.000, C 0.000 }
gfCNCPoint2[16817] = {X 121.2520, Y 99.8050, Z -3.0000, A 0.000, B 0.000, C 0.000 }
gfCNCPoint2[16818] = {X 120.9443, Y 98.9257, Z -3.0000, A 0.000, B 0.000, C 0.000 }
gfCNCPoint2[16819] = {X 120.8400, Y 98.0000, Z -3.0000, A 0.000, B 0.000, C 0.000 }
gfCNCPoint2[16820] = {X 120.8400, Y 97.0659, Z -3.0000, A 0.000, B 0.000, C 0.000 }
gfCNCPoint2[16821] = {X 120.9406, Y 96.1566, Z -3.0000, A 0.000, B 0.000, C 0.000 }
gfCNCPoint2[16822] = {X 121.2376, Y 95.2912, Z -3.0000, A 0.000, B 0.000, C 0.000 }
gfCNCPoint2[16823] = {X 121.7165, Y 94.5116, Z -3.0000, A 0.000, B 0.000, C 0.000 }
gfCNCPoint2[16824] = {X 122.3543, Y 93.8556, Z -3.0000, A 0.000, B 0.000, C 0.000 }
gfCNCPoint2[16825] = {X 123.1201, Y 93.3549, Z -3.0000, A 0.000, B 0.000, C 0.000 }
gfCNCPoint2[16826] = {X 123.9768, Y 93.0337, Z -3.0000, A 0.000, B 0.000, C 0.000 }
gfCNCPoint2[16827] = {X 124.8830, Y 92.9076, Z -3.0000, A 0.000, B 0.000, C 0.000 }
gfCNCPoint2[16828] = {X 124.9156, Y 92.8900, Z -3.0000, A 0.000, B 0.000, C 0.000 }
gfCNCPoint2[16829] = {X 124.9514, Y 92.8804, Z -3.0000, A 0.000, B 0.000, C 0.000 }
gfCNCPoint2[16830] = {X 125.4716, Y 92.8032, Z -3.0000, A 0.000, B 0.000, C 0.000 }
gfCNCPoint2[16831] = {X 126.3314, Y 92.6572, Z -3.0000, A 0.000, B 0.000, C 0.000 }
gfCNCPoint2[16832] = {X 127.1792, Y 92.4525, Z -3.0000, A 0.000, B 0.000, C 0.000 }
gfCNCPoint2[16833] = {X 128.4218, Y 91.2831, Z -3.0000, A 0.000, B 0.000, C 0.000 }
gfCNCPoint2[16834] = {X 129.5985, Y 90.0473, Z -3.0000, A 0.000, B 0.000, C 0.000 }
gfCNCPoint2[16835] = {X 140.7987, Y 77.7480, Z -3.0000, A 0.000, B 0.000, C 0.000 }
gfCNCPoint2[16836] = {X 137.8412, Y 75.0548, Z -3.0000, A 0.000, B 0.000, C 0.000 }
gfCNCPoint2[16837] = {X 140.8578, Y 77.8019, Z -3.0000, A 0.000, B 0.000, C 0.000 }
gfCNCPoint2[16838] = {X 155.9353, Y 61.2447, Z -3.0000, A 0.000, B 0.000, C 0.000 }
gfCNCPoint2[16839] = {X 155.5466, Y 60.5384, Z -3.0000, A 0.000, B 0.000, C 0.000 }
